C01812=1027.852,290.719,373.173,170.734,46.693,159.011
C01813=1027.858,290.967,373.141,170.739,46.692,159.011
C01814=1027.865,291.215,373.110,170.743,46.691,159.011
C01815=1027.872,291.462,373.078,170.747,46.690,159.011
C01816=1027.883,291.868,373.026,170.754,46.689,159.012
C01817=1027.894,292.273,372.973,170.761,46.687,159.012
C01818=1027.906,292.679,372.921,170.769,46.685,159.013
C01819=1027.917,293.084,372.868,170.776,46.684,159.014
C01820=1027.923,293.332,372.837,170.781,46.683,159.014
C01821=1027.930,293.579,372.804,170.785,46.682,159.014
C01822=1027.937,293.828,372.772,170.789,46.681,159.015
C01823=1027.944,294.075,372.740,170.794,46.680,159.015
C01824=1027.950,294.323,372.707,170.798,46.679,159.015
C01825=1027.957,294.571,372.676,170.803,46.679,159.016
C01826=1027.963,294.818,372.643,170.807,46.678,159.016
C01827=1027.970,295.066,372.610,170.812,46.677,159.016
C01828=1027.977,295.314,372.578,170.816,46.676,159.017
C01829=1027.983,295.562,372.546,170.821,46.675,159.017
C01830=1027.990,295.810,372.513,170.826,46.675,159.018
C01831=1027.997,296.058,372.481,170.830,46.674,159.018
C01832=1028.003,296.305,372.448,170.834,46.673,159.018
C01833=1028.010,296.553,372.415,170.838,46.672,159.019
C01834=1028.017,296.800,372.383,170.844,46.671,159.019
C01835=1028.024,297.048,372.350,170.848,46.671,159.019
C01836=1028.030,297.297,372.318,170.852,46.670,159.020
C01837=1028.037,297.544,372.286,170.857,46.669,159.020
C01838=1028.043,297.791,372.253,170.861,46.668,159.020
C01839=1028.050,298.040,372.220,170.866,46.668,159.021
C01840=1028.057,298.287,372.188,170.871,46.667,159.021
C01841=1028.063,298.535,372.155,170.875,46.666,159.022
C01842=1028.070,298.783,372.122,170.879,46.666,159.022
C01843=1028.077,299.030,372.090,170.885,46.665,159.023
C01844=1028.083,299.278,372.057,170.889,46.665,159.023
C01845=1028.090,299.526,372.024,170.893,46.663,159.023
C01846=1028.097,299.773,371.992,170.898,46.663,159.024
C01847=1028.104,300.021,371.959,170.903,46.662,159.024
C01848=1028.111,300.269,371.926,170.908,46.661,159.024
C01849=1028.118,300.517,371.894,170.912,46.661,159.025
C01850=1028.125,300.764,371.860,170.917,46.660,159.025
C01851=1028.131,301.012,371.827,170.922,46.659,159.026
C01852=1028.138,301.259,371.795,170.926,46.659,159.026
C01853=1028.145,301.507,371.762,170.930,46.658,159.026
C01854=1028.151,301.755,371.729,170.936,46.657,159.027
C01855=1028.159,302.003,371.697,170.940,46.657,159.027
C01856=1028.165,302.251,371.664,170.945,46.656,159.028
C01857=1028.172,302.498,371.630,170.950,46.656,159.028
C01858=1028.179,302.746,371.597,170.954,46.655,159.029
C01859=1028.186,302.994,371.565,170.959,46.654,159.029
C01860=1028.193,303.241,371.532,170.963,46.654,159.029
C01861=1028.200,303.489,371.498,170.969,46.653,159.030
C01862=1028.207,303.736,371.466,170.973,46.652,159.030
C01863=1028.214,303.985,371.433,170.978,46.652,159.031
C01864=1028.220,304.232,371.399,170.983,46.651,159.031
C01865=1028.228,304.480,371.367,170.987,46.651,159.032
C01866=1028.234,304.727,371.334,170.992,46.650,159.032
C01867=1028.241,304.975,371.300,170.996,46.649,159.032
C01868=1028.249,305.222,371.268,171.002,46.648,159.033
C01869=1028.255,305.470,371.235,171.006,46.648,159.033
C01870=1028.263,305.718,371.201,171.011,46.647,159.034
C01871=1028.269,305.966,371.169,171.016,46.647,159.034
C01872=1028.275,306.176,371.140,171.020,46.646,159.035
C01873=1028.281,306.388,371.112,171.024,46.646,159.035
C01874=1028.287,306.599,371.083,171.029,46.646,159.036
C01875=1028.293,306.810,371.056,171.032,46.645,159.036
C01876=1028.300,307.022,371.027,171.036,46.644,159.036
C01877=1028.305,307.233,370.999,171.040,46.644,159.037
C01878=1028.312,307.445,370.970,171.045,46.644,159.037
C01879=1028.318,307.656,370.943,171.049,46.643,159.037
C01880=1028.325,307.904,370.909,171.053,46.643,159.038
C01881=1028.331,308.151,370.876,171.059,46.642,159.038
C01882=1028.339,308.398,370.843,171.063,46.642,159.039
C01883=1028.346,308.647,370.810,171.068,46.641,159.039
C01884=1028.353,308.894,370.776,171.073,46.641,159.040
C01885=1028.360,309.141,370.742,171.078,46.640,159.040
C01886=1028.367,309.389,370.710,171.083,46.640,159.041
C01887=1028.375,309.637,370.676,171.088,46.639,159.041
C01888=1028.381,309.884,370.643,171.092,46.639,159.042
C01889=1028.388,310.132,370.610,171.098,46.638,159.042
C01890=1028.396,310.380,370.576,171.102,46.638,159.043
C01891=1028.403,310.627,370.542,171.107,46.637,159.043
C01892=1028.410,310.875,370.510,171.112,46.637,159.044
C01893=1028.417,311.123,370.476,171.117,46.636,159.044
C01894=1028.424,311.370,370.442,171.122,46.636,159.045
C01895=1028.430,311.618,370.408,171.127,46.636,159.045
C01896=1028.437,311.865,370.374,171.132,46.635,159.046
C01897=1028.444,312.113,370.340,171.137,46.635,159.046
C01898=1028.451,312.361,370.307,171.142,46.635,159.047
C01899=1028.458,312.607,370.272,171.147,46.635,159.047
C01900=1028.465,312.855,370.238,171.151,46.634,159.048
C01901=1028.472,313.103,370.204,171.157,46.634,159.049
C01902=1028.478,313.351,370.170,171.161,46.634,159.049
C01903=1028.486,313.598,370.136,171.167,46.634,159.050
C01904=1028.492,313.845,370.102,171.171,46.633,159.050
C01905=1028.499,314.093,370.068,171.177,46.633,159.051
C01906=1028.506,314.341,370.034,171.181,46.633,159.051
C01907=1028.513,314.588,369.999,171.187,46.633,159.052
C01908=1028.520,314.836,369.965,171.192,46.633,159.052
C01909=1028.526,315.083,369.932,171.197,46.632,159.053
C01910=1028.533,315.331,369.897,171.202,46.633,159.054
C01911=1028.540,315.578,369.863,171.207,46.632,159.054
C01912=1028.548,315.826,369.829,171.213,46.632,159.055
C01913=1028.554,316.074,369.795,171.217,46.632,159.055
C01914=1028.561,316.321,369.761,171.223,46.631,159.056
C01915=1028.569,316.568,369.726,171.227,46.631,159.056
C01916=1028.575,316.816,369.692,171.233,46.631,159.057
C01917=1028.582,317.064,369.658,171.237,46.631,159.057
C01918=1028.590,317.311,369.623,171.243,46.631,159.058
C01919=1028.596,317.559,369.589,171.248,46.631,159.059
C01920=1028.604,317.806,369.554,171.253,46.630,159.059
C01921=1028.611,318.053,369.521,171.258,46.630,159.060
C01922=1028.617,318.301,369.487,171.263,46.630,159.060
C01923=1028.624,318.548,369.452,171.269,46.630,159.061
C01924=1028.632,318.797,369.417,171.273,46.630,159.062
C01925=1028.639,319.044,369.383,171.279,46.630,159.062
C01926=1028.646,319.292,369.349,171.284,46.630,159.063
C01927=1028.653,319.539,369.314,171.289,46.630,159.063
C01928=1028.660,319.787,369.280,171.294,46.629,159.064
C01929=1028.668,320.034,369.245,171.300,46.629,159.065
C01930=1028.674,320.282,369.211,171.304,46.629,159.065
C01931=1028.682,320.529,369.176,171.310,46.629,159.066
C01932=1028.688,320.743,369.146,171.315,46.629,159.066
C01933=1028.694,320.957,369.116,171.319,46.629,159.067
C01934=1028.700,321.170,369.087,171.324,46.629,159.068
C01935=1028.706,321.384,369.057,171.328,46.629,159.068
C01936=1028.712,321.597,369.027,171.333,46.629,159.069
C01937=1028.719,321.811,368.997,171.337,46.629,159.069
C01938=1028.725,322.025,368.967,171.342,46.629,159.070
C01939=1028.731,322.239,368.937,171.346,46.629,159.070
C01940=1028.739,322.486,368.903,171.352,46.629,159.071
C01941=1028.746,322.733,368.868,171.356,46.629,159.071
C01942=1028.753,322.981,368.834,171.362,46.629,159.072
C01943=1028.760,323.229,368.799,171.368,46.629,159.073
C01944=1028.767,323.477,368.764,171.373,46.629,159.073
C01945=1028.775,323.724,368.729,171.378,46.629,159.074
C01946=1028.782,323.971,368.695,171.384,46.629,159.075
C01947=1028.789,324.219,368.660,171.389,46.629,159.075
C01948=1028.797,324.466,368.625,171.394,46.629,159.076
C01949=1028.804,324.714,368.590,171.399,46.629,159.077
C01950=1028.811,324.961,368.555,171.405,46.629,159.077
C01951=1028.819,325.209,368.521,171.411,46.629,159.078
C01952=1028.826,325.456,368.485,171.415,46.629,159.079
C01953=1028.834,325.703,368.451,171.421,46.629,159.079
C01954=1028.841,325.951,368.415,171.427,46.629,159.080
C01955=1028.849,326.198,368.381,171.433,46.629,159.081
C01956=1028.855,326.446,368.346,171.437,46.629,159.081
C01957=1028.863,326.693,368.311,171.443,46.629,159.082
C01958=1028.871,326.940,368.276,171.448,46.629,159.083
C01959=1028.878,327.188,368.241,171.454,46.629,159.083
C01960=1028.886,327.435,368.206,171.459,46.630,159.084
C01961=1028.893,327.683,368.171,171.465,46.630,159.085
C01962=1028.900,327.931,368.136,171.470,46.630,159.085
C01963=1028.907,328.178,368.101,171.476,46.630,159.086
C01964=1028.915,328.425,368.065,171.481,46.630,159.087
C01965=1028.922,328.673,368.030,171.486,46.630,159.087
C01966=1028.929,328.920,367.995,171.492,46.631,159.088
C01967=1028.936,329.167,367.959,171.498,46.631,159.089
C01968=1028.943,329.415,367.923,171.503,46.632,159.090
C01969=1028.951,329.662,367.889,171.509,46.632,159.090
C01970=1028.958,329.909,367.852,171.515,46.632,159.091
C01971=1028.965,330.157,367.817,171.520,46.632,159.092
C01972=1028.973,330.404,367.781,171.526,46.632,159.093
C01973=1028.980,330.652,367.746,171.531,46.633,159.093
C01974=1028.987,330.899,367.710,171.537,46.633,159.094
C01975=1028.994,331.146,367.675,171.542,46.633,159.095
C01976=1029.002,331.394,367.639,171.548,46.634,159.096
C01977=1029.009,331.641,367.604,171.554,46.633,159.096
C01978=1029.017,331.888,367.568,171.559,46.634,159.097
C01979=1029.024,332.136,367.532,171.565,46.635,159.098
C01980=1029.031,332.383,367.496,171.570,46.635,159.099
C01981=1029.038,332.631,367.461,171.576,46.635,159.100
C01982=1029.046,332.878,367.425,171.582,46.636,159.100
C01983=1029.054,333.124,367.390,171.588,46.636,159.101
C01984=1029.061,333.372,367.354,171.593,46.636,159.102
C01985=1029.069,333.620,367.318,171.599,46.637,159.103
C01986=1029.076,333.867,367.282,171.604,46.637,159.103
C01987=1029.083,334.115,367.247,171.610,46.637,159.104
C01988=1029.091,334.362,367.210,171.616,46.638,159.105
C01989=1029.098,334.609,367.175,171.622,46.638,159.106
C01990=1029.105,334.856,367.138,171.627,46.639,159.106
C01991=1029.113,335.103,367.102,171.633,46.639,159.107
C01992=1029.119,335.315,367.071,171.638,46.640,159.108
C01993=1029.125,335.527,367.041,171.643,46.640,159.109
C01994=1029.131,335.738,367.009,171.648,46.641,159.109
C01995=1029.137,335.950,366.978,171.653,46.641,159.110
C01996=1029.144,336.162,366.948,171.658,46.642,159.111
C01997=1029.150,336.372,366.916,171.662,46.642,159.111
C01998=1029.156,336.584,366.886,171.668,46.642,159.112
C01999=1029.163,336.796,366.855,171.673,46.642,159.113
C02000=1029.170,337.043,366.818,171.679,46.643,159.114
C02001=1029.178,337.290,366.782,171.685,46.643,159.115
C02002=1029.185,337.537,366.746,171.690,46.644,159.115
C02003=1029.193,337.785,366.710,171.696,46.645,159.116
C02004=1029.200,338.032,366.674,171.701,46.645,159.117
C02005=1029.208,338.279,366.638,171.707,46.646,159.118
C02006=1029.215,338.527,366.601,171.713,46.646,159.119
C02007=1029.222,338.774,366.565,171.719,46.647,159.120
C02008=1029.230,339.022,366.528,171.725,46.648,159.121
C02009=1029.238,339.269,366.491,171.731,46.648,159.121
C02010=1029.245,339.515,366.456,171.737,46.649,159.122
C02011=1029.253,339.763,366.419,171.743,46.649,159.123
C02012=1029.260,340.010,366.383,171.749,46.650,159.124
C02013=1029.268,340.257,366.346,171.755,46.650,159.125
C02014=1029.275,340.505,366.309,171.761,46.651,159.126
C02015=1029.283,340.752,366.273,171.767,46.652,159.127
C02016=1029.291,340.999,366.236,171.773,46.653,159.128
C02017=1029.297,341.246,366.200,171.779,46.653,159.128
C02018=1029.305,341.493,366.163,171.785,46.654,159.129
C02019=1029.313,341.740,366.127,171.791,46.655,159.130
C02020=1029.320,341.987,366.089,171.797,46.655,159.131
C02021=1029.328,342.235,366.053,171.803,46.656,159.132
C02022=1029.335,342.482,366.015,171.809,46.657,159.133
C02023=1029.343,342.730,365.979,171.815,46.657,159.134
C02024=1029.351,342.976,365.942,171.822,46.658,159.135
C02025=1029.358,343.223,365.905,171.827,46.659,159.136
C02026=1029.366,343.471,365.868,171.834,46.660,159.137
C02027=1029.373,343.718,365.831,171.840,46.661,159.138
C02028=1029.381,343.965,365.794,171.846,46.662,159.139
C02029=1029.389,344.212,365.758,171.852,46.662,159.139
C02030=1029.396,344.459,365.720,171.858,46.663,159.140
C02031=1029.404,344.706,365.683,171.864,46.664,159.141
C02032=1029.411,344.953,365.646,171.870,46.665,159.142
C02033=1029.419,345.201,365.610,171.876,46.665,159.143
C02034=1029.426,345.448,365.572,171.882,46.666,159.144
C02035=1029.434,345.695,365.535,171.889,46.668,159.145
C02036=1029.441,345.942,365.498,171.895,46.668,159.146
C02037=1029.450,346.189,365.460,171.901,46.669,159.147
C02038=1029.457,346.437,365.423,171.908,46.670,159.148
C02039=1029.465,346.683,365.386,171.914,46.671,159.149
C02040=1029.472,346.931,365.348,171.920,46.672,159.150
C02041=1029.480,347.177,365.311,171.926,46.673,159.151
C02042=1029.488,347.425,365.274,171.932,46.673,159.152
C02043=1029.496,347.672,365.237,171.939,46.674,159.153
C02044=1029.503,347.919,365.199,171.945,46.675,159.154
C02045=1029.511,348.166,365.162,171.951,46.677,159.155
C02046=1029.519,348.413,365.125,171.958,46.677,159.156
C02047=1029.527,348.660,365.088,171.964,46.678,159.157
C02048=1029.534,348.908,365.050,171.970,46.679,159.158
C02049=1029.542,349.154,365.011,171.977,46.680,159.159
C02050=1029.550,349.401,364.975,171.983,46.681,159.160
C02051=1029.557,349.648,364.937,171.989,46.682,159.161
C02052=1029.563,349.858,364.905,171.995,46.683,159.162
C02053=1029.570,350.068,364.873,172.000,46.684,159.163
C02054=1029.577,350.279,364.840,172.006,46.685,159.164
C02055=1029.584,350.488,364.809,172.011,46.686,159.165
C02056=1029.590,350.699,364.776,172.016,46.687,159.165
C02057=1029.597,350.908,364.745,172.023,46.688,159.166
C02058=1029.603,351.118,364.712,172.027,46.689,159.167
C02059=1029.610,351.328,364.680,172.034,46.690,159.168
C02060=1029.618,351.576,364.642,172.040,46.691,159.169
C02061=1029.625,351.822,364.604,172.046,46.692,159.170
C02062=1029.633,352.069,364.567,172.052,46.693,159.171
C02063=1029.641,352.316,364.529,172.059,46.694,159.172
C02064=1029.649,352.563,364.491,172.066,46.695,159.173
C02065=1029.656,352.810,364.453,172.072,46.696,159.174
C02066=1029.665,353.057,364.415,172.079,46.698,159.176
C02067=1029.672,353.304,364.377,172.085,46.699,159.177
C02068=1029.680,353.551,364.339,172.092,46.700,159.178
C02069=1029.688,353.798,364.301,172.098,46.701,159.179
C02070=1029.696,354.045,364.263,172.105,46.702,159.180
C02071=1029.704,354.292,364.225,172.112,46.703,159.181
C02072=1029.712,354.539,364.186,172.118,46.704,159.182
C02073=1029.720,354.786,364.149,172.125,46.706,159.183
C02074=1029.728,355.033,364.110,172.131,46.707,159.184
C02075=1029.736,355.279,364.073,172.138,46.708,159.185
C02076=1029.744,355.527,364.034,172.145,46.710,159.187
C02077=1029.752,355.773,363.996,172.151,46.711,159.188
C02078=1029.760,356.020,363.957,172.159,46.712,159.189
C02079=1029.767,356.267,363.919,172.165,46.713,159.190
C02080=1029.776,356.514,363.880,172.171,46.715,159.191
C02081=1029.784,356.761,363.842,172.179,46.716,159.192
C02082=1029.791,357.008,363.803,172.185,46.717,159.193
C02083=1029.799,357.255,363.765,172.191,46.718,159.194
C02084=1029.807,357.501,363.727,172.199,46.720,159.196
C02085=1029.815,357.749,363.688,172.206,46.721,159.197
C02086=1029.823,357.996,363.649,172.213,46.722,159.198
C02087=1029.831,358.242,363.611,172.219,46.724,159.199
C02088=1029.839,358.490,363.573,172.226,46.726,159.200
C02089=1029.847,358.737,363.534,172.233,46.726,159.202
C02090=1029.855,358.983,363.495,172.240,46.728,159.203
C02091=1029.863,359.230,363.456,172.247,46.730,159.204
C02092=1029.871,359.477,363.418,172.254,46.731,159.205
C02093=1029.879,359.724,363.379,172.260,46.732,159.206
C02094=1029.887,359.970,363.340,172.268,46.734,159.208
C02095=1029.895,360.218,363.302,172.274,46.735,159.209
C02096=1029.904,360.464,363.262,172.282,46.737,159.210
C02097=1029.912,360.711,363.224,172.288,46.738,159.211
C02098=1029.920,360.958,363.185,172.296,46.740,159.212
C02099=1029.927,361.205,363.145,172.302,46.741,159.214
C02100=1029.935,361.452,363.107,172.310,46.743,159.215
C02101=1029.944,361.699,363.068,172.316,46.745,159.216
C02102=1029.952,361.945,363.028,172.323,46.746,159.217
C02103=1029.959,362.192,362.989,172.330,46.748,159.219
C02104=1029.968,362.439,362.950,172.337,46.749,159.220
C02105=1029.976,362.685,362.911,172.344,46.751,159.221
C02106=1029.983,362.933,362.871,172.351,46.752,159.222
C02107=1029.992,363.179,362.832,172.359,46.754,159.224
C02108=1030.000,363.426,362.793,172.365,46.756,159.225
C02109=1030.008,363.673,362.753,172.373,46.757,159.226
C02110=1030.016,363.920,362.714,172.380,46.759,159.228
C02111=1030.025,364.167,362.675,172.387,46.760,159.229
C02112=1030.032,364.379,362.641,172.394,46.762,159.230
C02113=1030.038,364.592,362.607,172.400,46.763,159.231
C02114=1030.046,364.805,362.572,172.405,46.765,159.232
C02115=1030.053,365.019,362.539,172.412,46.766,159.233
C02116=1030.060,365.232,362.505,172.418,46.768,159.234
C02117=1030.067,365.445,362.471,172.425,46.769,159.236
C02118=1030.075,365.658,362.436,172.431,46.770,159.237
C02119=1030.081,365.871,362.402,172.437,46.772,159.238
C02120=1030.089,366.118,362.363,172.444,46.774,159.239
C02121=1030.098,366.364,362.323,172.452,46.776,159.241
C02122=1030.106,366.611,362.283,172.458,46.777,159.242
C02123=1030.114,366.858,362.244,172.466,46.779,159.243
C02124=1030.123,367.104,362.205,172.474,46.781,159.245
C02125=1030.131,367.352,362.165,172.481,46.783,159.246
C02126=1030.140,367.598,362.124,172.488,46.784,159.247
C02127=1030.148,367.845,362.085,172.496,46.786,159.249
C02128=1030.156,368.092,362.045,172.503,46.788,159.250
C02129=1030.164,368.338,362.006,172.510,46.790,159.251
C02130=1030.173,368.584,361.966,172.518,46.792,159.253
C02131=1030.181,368.832,361.926,172.525,46.794,159.254
C02132=1030.190,369.078,361.886,172.533,46.796,159.256
C02133=1030.199,369.324,361.846,172.541,46.798,159.257
C02134=1030.206,369.571,361.806,172.548,46.800,159.258
C02135=1030.214,369.817,361.766,172.555,46.801,159.260
C02136=1030.223,370.065,361.726,172.563,46.803,159.261
C02137=1030.231,370.311,361.685,172.571,46.805,159.263
C02138=1030.239,370.558,361.645,172.578,46.807,159.264
C02139=1030.248,370.804,361.605,172.585,46.809,159.265
C02140=1030.256,371.051,361.564,172.593,46.811,159.267
C02141=1030.265,371.297,361.525,172.601,46.813,159.268
C02142=1030.273,371.544,361.484,172.608,46.815,159.270
C02143=1030.282,371.791,361.443,172.616,46.817,159.271
C02144=1030.290,372.037,361.403,172.624,46.819,159.273
C02145=1030.298,372.283,361.363,172.632,46.821,159.274
C02146=1030.307,372.531,361.322,172.639,46.823,159.276
C02147=1030.315,372.777,361.282,172.646,46.825,159.277
C02148=1030.323,373.023,361.242,172.654,46.827,159.279
C02149=1030.332,373.270,361.201,172.662,46.829,159.280
C02150=1030.341,373.516,361.161,172.670,46.832,159.282
C02151=1030.350,373.763,361.120,172.678,46.834,159.283
C02152=1030.358,374.009,361.079,172.686,46.836,159.285
C02153=1030.367,374.256,361.039,172.694,46.838,159.286
C02154=1030.375,374.502,360.998,172.701,46.841,159.288
C02155=1030.384,374.749,360.957,172.709,46.843,159.289
C02156=1030.392,374.995,360.917,172.717,46.844,159.291
C02157=1030.401,375.242,360.876,172.724,46.846,159.292
C02158=1030.409,375.488,360.835,172.733,46.849,159.294
C02159=1030.418,375.735,360.795,172.741,46.851,159.295
C02160=1030.427,375.981,360.754,172.749,46.853,159.297
C02161=1030.435,376.228,360.713,172.757,46.855,159.298
C02162=1030.445,376.474,360.672,172.765,46.858,159.300
C02163=1030.453,376.721,360.632,172.773,46.860,159.301
C02164=1030.462,376.967,360.590,172.781,46.862,159.303
C02165=1030.471,377.214,360.549,172.789,46.864,159.305
C02166=1030.479,377.460,360.509,172.797,46.867,159.306
C02167=1030.488,377.706,360.467,172.805,46.869,159.308
C02168=1030.497,377.953,360.426,172.813,46.871,159.309
C02169=1030.505,378.199,360.385,172.821,46.874,159.311
C02170=1030.514,378.445,360.343,172.829,46.876,159.313
C02171=1030.522,378.692,360.302,172.837,46.878,159.314
C02172=1030.530,378.915,360.265,172.844,46.881,159.316
C02173=1030.538,379.139,360.227,172.852,46.883,159.317
C02174=1030.546,379.363,360.189,172.859,46.885,159.319
C02175=1030.553,379.586,360.152,172.867,46.887,159.320
C02176=1030.561,379.810,360.114,172.874,46.890,159.322
C02177=1030.570,380.034,360.076,172.882,46.892,159.323
C02178=1030.578,380.258,360.039,172.889,46.894,159.325
C02179=1030.586,380.480,360.001,172.897,46.896,159.326
C02180=1030.594,380.727,359.960,172.905,46.899,159.328
C02181=1030.603,380.974,359.918,172.913,46.901,159.330
C02182=1030.612,381.220,359.876,172.921,46.904,159.331
C02183=1030.621,381.466,359.835,172.930,46.906,159.333
C02184=1030.630,381.713,359.793,172.938,46.909,159.334
C02185=1030.639,381.959,359.751,172.947,46.911,159.336
C02186=1030.647,382.206,359.709,172.955,46.914,159.338
C02187=1030.656,382.452,359.667,172.963,46.916,159.340
C02188=1030.665,382.699,359.625,172.972,46.919,159.341
C02189=1030.674,382.944,359.583,172.980,46.922,159.343
C02190=1030.683,383.191,359.541,172.989,46.924,159.345
C02191=1030.692,383.437,359.500,172.997,46.926,159.346
C02192=1030.701,383.683,359.458,173.006,46.929,159.348
C02193=1030.710,383.930,359.416,173.014,46.932,159.350
C02194=1030.719,384.175,359.374,173.023,46.934,159.352
C02195=1030.728,384.422,359.332,173.032,46.937,159.354
C02196=1030.737,384.668,359.290,173.040,46.940,159.355
C02197=1030.746,384.914,359.248,173.048,46.943,159.357
C02198=1030.755,385.160,359.206,173.058,46.945,159.359
C02199=1030.765,385.406,359.164,173.066,46.948,159.361
C02200=1030.774,385.652,359.122,173.074,46.950,159.362
C02201=1030.783,385.899,359.079,173.084,46.953,159.364
C02202=1030.792,386.145,359.038,173.092,46.956,159.366
C02203=1030.802,386.391,358.995,173.101,46.959,159.368
C02204=1030.810,386.637,358.953,173.110,46.962,159.370
C02205=1030.820,386.884,358.911,173.118,46.964,159.371
C02206=1030.829,387.130,358.868,173.128,46.967,159.373
C02207=1030.838,387.376,358.826,173.136,46.970,159.375
C02208=1030.847,387.622,358.783,173.145,46.973,159.377
C02209=1030.857,387.868,358.741,173.154,46.976,159.379
C02210=1030.865,388.114,358.698,173.163,46.979,159.381
C02211=1030.875,388.360,358.655,173.172,46.981,159.383
C02212=1030.884,388.607,358.612,173.181,46.985,159.384
C02213=1030.893,388.853,358.569,173.189,46.988,159.386
C02214=1030.902,389.098,358.527,173.199,46.990,159.388
C02215=1030.912,389.345,358.484,173.207,46.993,159.390
C02216=1030.920,389.591,358.441,173.217,46.996,159.392
C02217=1030.930,389.837,358.399,173.225,46.999,159.394
C02218=1030.940,390.083,358.356,173.235,47.002,159.396
C02219=1030.948,390.329,358.313,173.243,47.005,159.398
C02220=1030.958,390.576,358.270,173.253,47.008,159.400
C02221=1030.967,390.821,358.226,173.262,47.011,159.402
C02222=1030.977,391.067,358.183,173.271,47.014,159.404
C02223=1030.985,391.314,358.140,173.281,47.017,159.406
C02224=1030.995,391.559,358.097,173.289,47.020,159.408
C02225=1031.004,391.805,358.054,173.299,47.023,159.409
C02226=1031.014,392.052,358.011,173.308,47.027,159.412
C02227=1031.023,392.297,357.968,173.317,47.029,159.413
C02228=1031.032,392.544,357.925,173.327,47.033,159.416
C02229=1031.042,392.790,357.881,173.336,47.036,159.417
C02230=1031.051,393.036,357.838,173.345,47.039,159.420
C02231=1031.061,393.281,357.794,173.355,47.042,159.421
C02232=1031.071,393.545,357.748,173.365,47.046,159.424
C02233=1031.081,393.811,357.701,173.375,47.049,159.426
C02234=1031.092,394.074,357.655,173.385,47.052,159.428
C02235=1031.101,394.338,357.608,173.395,47.056,159.430
C02236=1031.111,394.584,357.563,173.405,47.060,159.432
C02237=1031.121,394.830,357.520,173.414,47.062,159.434
C02238=1031.130,395.076,357.476,173.424,47.066,159.436
C02239=1031.139,395.322,357.433,173.433,47.069,159.439
C02240=1031.149,395.568,357.389,173.443,47.072,159.441
C02241=1031.158,395.814,357.345,173.453,47.076,159.443
C02242=1031.168,396.061,357.301,173.462,47.079,159.445
C02243=1031.178,396.306,357.257,173.471,47.083,159.447
C02244=1031.187,396.551,357.213,173.481,47.086,159.449
C02245=1031.197,396.797,357.169,173.491,47.089,159.451
C02246=1031.207,397.043,357.125,173.501,47.093,159.454
C02247=1031.216,397.289,357.081,173.511,47.096,159.456
C02248=1031.225,397.521,357.040,173.520,47.099,159.457
C02249=1031.235,397.753,356.998,173.529,47.103,159.460
C02250=1031.244,397.986,356.956,173.538,47.106,159.462
C02251=1031.253,398.218,356.915,173.548,47.109,159.464
C02252=1031.262,398.450,356.873,173.557,47.112,159.466
C02253=1031.271,398.682,356.831,173.566,47.116,159.468
C02254=1031.280,398.914,356.790,173.576,47.119,159.470
C02255=1031.290,399.145,356.747,173.585,47.122,159.472
C02256=1031.300,399.392,356.703,173.595,47.126,159.474
C02257=1031.309,399.637,356.658,173.605,47.130,159.476
C02258=1031.319,399.883,356.614,173.615,47.133,159.479
C02259=1031.329,400.128,356.570,173.625,47.137,159.481
C02260=1031.339,400.374,356.525,173.635,47.140,159.483
C02261=1031.348,400.620,356.481,173.646,47.144,159.486
C02262=1031.359,400.866,356.436,173.655,47.147,159.488
C02263=1031.368,401.112,356.391,173.666,47.151,159.490
C02264=1031.378,401.357,356.346,173.676,47.155,159.492
C02265=1031.388,401.603,356.302,173.686,47.159,159.495
C02266=1031.398,401.849,356.256,173.697,47.162,159.497
C02267=1031.408,402.095,356.211,173.707,47.166,159.499
C02268=1031.417,402.340,356.167,173.717,47.170,159.502
C02269=1031.427,402.586,356.122,173.728,47.174,159.504
C02270=1031.438,402.832,356.077,173.738,47.178,159.506
C02271=1031.447,403.077,356.032,173.748,47.182,159.509
C02272=1031.457,403.323,355.987,173.759,47.185,159.511
C02273=1031.468,403.568,355.941,173.769,47.189,159.513
C02274=1031.477,403.814,355.896,173.779,47.193,159.516
C02275=1031.488,404.060,355.851,173.790,47.197,159.518
C02276=1031.498,404.305,355.806,173.800,47.201,159.521
C02277=1031.507,404.551,355.761,173.811,47.204,159.523
C02278=1031.518,404.797,355.716,173.822,47.209,159.525
C02279=1031.527,405.042,355.669,173.832,47.212,159.528
C02280=1031.537,405.288,355.624,173.843,47.216,159.530
C02281=1031.548,405.534,355.578,173.854,47.220,159.533
C02282=1031.558,405.779,355.533,173.864,47.224,159.535
C02283=1031.568,406.025,355.488,173.875,47.228,159.538
C02284=1031.578,406.270,355.442,173.886,47.232,159.540
C02285=1031.589,406.516,355.397,173.896,47.236,159.542
C02286=1031.599,406.762,355.351,173.908,47.240,159.545
C02287=1031.609,407.006,355.305,173.918,47.245,159.548
C02288=1031.619,407.252,355.259,173.929,47.248,159.550
C02289=1031.629,407.499,355.214,173.940,47.252,159.553
C02290=1031.640,407.744,355.168,173.951,47.256,159.555
C02291=1031.650,407.989,355.122,173.962,47.261,159.558
C02292=1031.661,408.247,355.074,173.973,47.265,159.560
C02293=1031.672,408.505,355.026,173.985,47.269,159.563
C02294=1031.683,408.763,354.977,173.997,47.273,159.566
C02295=1031.694,409.021,354.929,174.009,47.278,159.568
C02296=1031.705,409.267,354.883,174.019,47.282,159.571
C02297=1031.716,409.512,354.837,174.031,47.286,159.574
C02298=1031.727,409.757,354.791,174.042,47.290,159.576
C02299=1031.736,410.003,354.744,174.053,47.295,159.579
C02300=1031.747,410.249,354.698,174.065,47.299,159.581
C02301=1031.758,410.495,354.652,174.076,47.303,159.584
C02302=1031.769,410.740,354.606,174.087,47.308,159.587
C02303=1031.778,410.985,354.559,174.098,47.312,159.589
C02304=1031.789,411.230,354.513,174.110,47.317,159.592
C02305=1031.799,411.476,354.466,174.121,47.321,159.595
C02306=1031.810,411.721,354.420,174.133,47.326,159.598
C02307=1031.821,411.966,354.373,174.144,47.329,159.600
C02308=1031.831,412.212,354.327,174.156,47.334,159.603
C02309=1031.842,412.457,354.280,174.167,47.339,159.606
C02310=1031.853,412.703,354.232,174.179,47.343,159.608
C02311=1031.864,412.948,354.186,174.190,47.347,159.611
C02312=1031.874,413.194,354.139,174.202,47.352,159.614
C02313=1031.884,413.439,354.093,174.214,47.356,159.617
C02314=1031.895,413.685,354.045,174.226,47.361,159.619
C02315=1031.906,413.930,353.998,174.238,47.366,159.622
C02316=1031.916,414.175,353.951,174.249,47.370,159.625
C02317=1031.927,414.420,353.905,174.261,47.375,159.628
C02318=1031.939,414.666,353.858,174.272,47.379,159.631
C02319=1031.949,414.911,353.810,174.284,47.384,159.633
C02320=1031.961,415.156,353.763,174.296,47.388,159.636
C02321=1031.971,415.401,353.715,174.308,47.393,159.639
C02322=1031.983,415.647,353.668,174.320,47.398,159.642
C02323=1031.993,415.892,353.621,174.333,47.402,159.645
C02324=1032.005,416.138,353.573,174.345,47.407,159.648
C02325=1032.015,416.383,353.526,174.357,47.412,159.651
C02326=1032.026,416.628,353.479,174.369,47.417,159.654
C02327=1032.037,416.874,353.431,174.381,47.421,159.657
C02328=1032.048,417.118,353.383,174.394,47.426,159.660
C02329=1032.059,417.364,353.336,174.405,47.431,159.662
C02330=1032.070,417.609,353.288,174.419,47.436,159.665
C02331=1032.081,417.854,353.240,174.431,47.441,159.668
C02332=1032.092,418.100,353.192,174.443,47.446,159.671
C02333=1032.103,418.345,353.145,174.455,47.451,159.675
C02334=1032.114,418.590,353.097,174.468,47.456,159.678
C02335=1032.125,418.835,353.048,174.481,47.460,159.681
C02336=1032.137,419.080,353.001,174.493,47.465,159.684
C02337=1032.148,419.325,352.953,174.505,47.470,159.687
C02338=1032.159,419.570,352.904,174.518,47.475,159.690
C02339=1032.170,419.816,352.856,174.531,47.480,159.693
C02340=1032.182,420.061,352.808,174.544,47.485,159.696
C02341=1032.193,420.306,352.760,174.556,47.490,159.699
C02342=1032.204,420.550,352.711,174.569,47.495,159.702
C02343=1032.215,420.796,352.663,174.582,47.500,159.705
C02344=1032.227,421.041,352.615,174.594,47.506,159.708
C02345=1032.238,421.285,352.566,174.608,47.510,159.711
C02346=1032.249,421.531,352.518,174.621,47.516,159.715
C02347=1032.260,421.776,352.470,174.634,47.521,159.718
C02348=1032.272,422.020,352.421,174.647,47.526,159.721
C02349=1032.284,422.267,352.373,174.659,47.531,159.724
C02350=1032.295,422.511,352.324,174.673,47.536,159.727
C02351=1032.307,422.756,352.275,174.686,47.541,159.731
C02352=1032.319,423.025,352.222,174.700,47.547,159.734
C02353=1032.332,423.293,352.169,174.715,47.552,159.738
C02354=1032.345,423.561,352.115,174.729,47.559,159.741
C02355=1032.357,423.829,352.062,174.744,47.564,159.745
C02356=1032.369,424.073,352.013,174.757,47.570,159.748
C02357=1032.380,424.318,351.964,174.771,47.575,159.751
C02358=1032.392,424.563,351.915,174.784,47.580,159.755
C02359=1032.404,424.808,351.864,174.798,47.586,159.758
C02360=1032.415,425.052,351.815,174.812,47.591,159.762
C02361=1032.427,425.297,351.766,174.825,47.596,159.765
C02362=1032.439,425.543,351.717,174.839,47.602,159.768
C02363=1032.450,425.787,351.668,174.852,47.607,159.772
C02364=1032.463,426.032,351.618,174.866,47.613,159.775
C02365=1032.474,426.277,351.569,174.879,47.618,159.778
C02366=1032.486,426.522,351.519,174.893,47.624,159.782
C02367=1032.498,426.767,351.470,174.908,47.629,159.785
C02368=1032.510,427.011,351.420,174.922,47.635,159.789
C02369=1032.521,427.256,351.371,174.936,47.640,159.792
C02370=1032.534,427.501,351.321,174.950,47.646,159.796
C02371=1032.546,427.746,351.270,174.964,47.652,159.799
C02372=1032.557,427.990,351.220,174.977,47.657,159.803
C02373=1032.569,428.236,351.171,174.992,47.664,159.806
C02374=1032.581,428.480,351.121,175.006,47.669,159.810
C02375=1032.593,428.725,351.071,175.021,47.675,159.814
C02376=1032.605,428.969,351.021,175.035,47.680,159.817
C02377=1032.617,429.215,350.970,175.049,47.686,159.821
C02378=1032.629,429.458,350.920,175.063,47.692,159.824
C02379=1032.641,429.703,350.870,175.078,47.697,159.828
C02380=1032.654,429.948,350.820,175.092,47.704,159.832
C02381=1032.665,430.193,350.769,175.107,47.709,159.835
C02382=1032.678,430.437,350.718,175.121,47.715,159.839
C02383=1032.690,430.682,350.668,175.136,47.721,159.843
C02384=1032.702,430.927,350.618,175.151,47.727,159.846
C02385=1032.715,431.171,350.567,175.165,47.733,159.850
C02386=1032.727,431.416,350.516,175.180,47.739,159.854
C02387=1032.739,431.660,350.466,175.194,47.745,159.857
C02388=1032.752,431.904,350.415,175.210,47.751,159.861
C02389=1032.764,432.149,350.365,175.225,47.756,159.865
C02390=1032.777,432.393,350.314,175.239,47.763,159.869
C02391=1032.789,432.638,350.262,175.255,47.769,159.873
C02392=1032.801,432.882,350.212,175.270,47.775,159.877
C02393=1032.814,433.127,350.162,175.285,47.781,159.880
C02394=1032.827,433.372,350.110,175.300,47.787,159.884
C02395=1032.839,433.616,350.060,175.316,47.793,159.888
C02396=1032.851,433.861,350.008,175.331,47.799,159.892
C02397=1032.865,434.105,349.956,175.347,47.805,159.896
C02398=1032.877,434.349,349.905,175.362,47.811,159.900
C02399=1032.889,434.594,349.854,175.378,47.817,159.904
C02400=1032.903,434.838,349.803,175.392,47.824,159.908
C02401=1032.915,435.082,349.751,175.408,47.830,159.912
C02402=1032.928,435.327,349.700,175.424,47.836,159.916
C02403=1032.941,435.571,349.648,175.439,47.843,159.920
C02404=1032.953,435.816,349.596,175.455,47.849,159.924
C02405=1032.966,436.060,349.545,175.472,47.855,159.928
C02406=1032.979,436.304,349.492,175.488,47.862,159.932
C02407=1032.992,436.548,349.441,175.503,47.868,159.936
C02408=1033.004,436.793,349.389,175.519,47.874,159.940
C02409=1033.018,437.037,349.337,175.535,47.881,159.944
C02410=1033.030,437.281,349.285,175.551,47.887,159.948
C02411=1033.044,437.525,349.233,175.568,47.894,159.952
C02412=1033.057,437.782,349.178,175.585,47.900,159.957
C02413=1033.071,438.040,349.123,175.601,47.908,159.961
C02414=1033.085,438.296,349.068,175.619,47.915,159.966
C02415=1033.098,438.553,349.013,175.636,47.921,159.970
C02416=1033.111,438.798,348.961,175.653,47.928,159.974
C02417=1033.125,439.042,348.909,175.669,47.934,159.978
C02418=1033.138,439.286,348.856,175.686,47.941,159.983
C02419=1033.151,439.531,348.804,175.702,47.948,159.987
C02420=1033.164,439.775,348.751,175.719,47.954,159.991
C02421=1033.177,440.018,348.697,175.735,47.961,159.996
C02422=1033.191,440.263,348.645,175.753,47.968,160.000
C02423=1033.204,440.507,348.592,175.770,47.975,160.004
C02424=1033.217,440.751,348.539,175.786,47.982,160.009
C02425=1033.231,440.994,348.486,175.803,47.988,160.013
C02426=1033.244,441.238,348.433,175.821,47.995,160.018
C02427=1033.258,441.483,348.380,175.838,48.002,160.022
C02428=1033.272,441.727,348.327,175.855,48.009,160.027
C02429=1033.285,441.971,348.274,175.871,48.015,160.031
C02430=1033.299,442.214,348.221,175.889,48.022,160.036
C02431=1033.312,442.459,348.168,175.906,48.029,160.040
C02432=1033.325,442.703,348.114,175.924,48.037,160.045
C02433=1033.339,442.946,348.061,175.941,48.044,160.049
C02434=1033.353,443.191,348.008,175.959,48.050,160.054
C02435=1033.367,443.434,347.954,175.977,48.057,160.058
C02436=1033.381,443.677,347.900,175.995,48.064,160.063
C02437=1033.395,443.919,347.848,176.012,48.071,160.068
C02438=1033.410,444.163,347.796,176.030,48.078,160.072
C02439=1033.425,444.407,347.743,176.049,48.085,160.077
C02440=1033.441,444.650,347.692,176.066,48.092,160.081
C02441=1033.457,444.894,347.641,176.085,48.098,160.086
C02442=1033.474,445.137,347.589,176.103,48.105,160.091
C02443=1033.492,445.381,347.539,176.120,48.111,160.095
C02444=1033.509,445.625,347.489,176.138,48.117,160.099
C02445=1033.527,445.869,347.439,176.157,48.124,160.104
C02446=1033.546,446.113,347.391,176.176,48.130,160.109
C02447=1033.566,446.358,347.341,176.195,48.136,160.113
C02448=1033.586,446.602,347.293,176.213,48.142,160.117
C02449=1033.606,446.845,347.246,176.232,48.148,160.122
C02450=1033.627,447.089,347.198,176.251,48.153,160.126
C02451=1033.648,447.335,347.151,176.270,48.160,160.131
C02452=1033.671,447.579,347.105,176.289,48.165,160.135
C02453=1033.693,447.823,347.058,176.308,48.171,160.140
C02454=1033.716,448.068,347.012,176.327,48.177,160.144
C02455=1033.739,448.313,346.967,176.346,48.182,160.149
C02456=1033.764,448.558,346.922,176.365,48.187,160.153
C02457=1033.788,448.802,346.877,176.385,48.192,160.158
C02458=1033.813,449.048,346.833,176.404,48.198,160.162
C02459=1033.838,449.293,346.790,176.424,48.203,160.166
C02460=1033.865,449.537,346.747,176.444,48.208,160.171
C02461=1033.891,449.783,346.705,176.463,48.213,160.175
C02462=1033.918,450.029,346.662,176.483,48.218,160.180
C02463=1033.946,450.273,346.620,176.503,48.223,160.184
C02464=1033.974,450.519,346.578,176.523,48.228,160.188
C02465=1034.003,450.765,346.537,176.544,48.232,160.193
C02466=1034.032,451.010,346.497,176.564,48.237,160.197
C02467=1034.062,451.255,346.457,176.583,48.242,160.201
C02468=1034.092,451.500,346.417,176.604,48.246,160.206
C02469=1034.122,451.747,346.377,176.625,48.250,160.210
C02470=1034.154,451.992,346.338,176.645,48.255,160.214
C02471=1034.185,452.237,346.300,176.666,48.259,160.219
C02472=1034.231,452.584,346.246,176.695,48.266,160.225
C02473=1034.278,452.931,346.194,176.725,48.271,160.231
C02474=1033.992,452.993,345.866,176.728,48.338,160.252
C02475=1033.949,452.671,345.914,176.701,48.333,160.247
C02476=1033.905,452.348,345.964,176.673,48.328,160.241
C02477=1033.874,452.102,346.002,176.652,48.323,160.237
C02478=1033.843,451.857,346.040,176.632,48.319,160.232
C02479=1033.811,451.612,346.080,176.611,48.315,160.228
C02480=1033.781,451.365,346.119,176.591,48.310,160.224
C02481=1033.751,451.120,346.159,176.570,48.306,160.219
C02482=1033.722,450.875,346.200,176.550,48.301,160.215
C02483=1033.693,450.629,346.240,176.530,48.297,160.211
C02484=1033.664,450.384,346.281,176.510,48.292,160.206
C02485=1033.637,450.139,346.323,176.490,48.287,160.202
C02486=1033.609,449.894,346.366,176.470,48.283,160.198
C02487=1033.582,449.648,346.408,176.450,48.278,160.193
C02488=1033.556,449.403,346.450,176.430,48.273,160.189
C02489=1033.529,449.158,346.494,176.410,48.268,160.184
C02490=1033.505,448.913,346.538,176.391,48.262,160.180
C02491=1033.479,448.668,346.582,176.371,48.257,160.175
C02492=1033.455,448.423,346.627,176.352,48.252,160.171
C02493=1033.432,448.178,346.672,176.333,48.247,160.167
C02494=1033.409,447.933,346.717,176.313,48.241,160.162
C02495=1033.386,447.690,346.764,176.294,48.236,160.158
C02496=1033.363,447.444,346.810,176.275,48.231,160.153
C02497=1033.342,447.200,346.857,176.256,48.224,160.149
C02498=1033.321,446.956,346.904,176.237,48.219,160.144
C02499=1033.300,446.711,346.952,176.218,48.213,160.140
C02500=1033.279,446.468,346.999,176.200,48.207,160.135
C02501=1033.260,446.223,347.048,176.180,48.202,160.131
C02502=1033.241,445.979,347.097,176.162,48.195,160.126
C02503=1033.222,445.735,347.146,176.144,48.189,160.122
C02504=1033.204,445.492,347.196,176.125,48.183,160.117
C02505=1033.186,445.247,347.246,176.107,48.177,160.113
C02506=1033.169,445.003,347.297,176.089,48.170,160.108
C02507=1033.152,444.759,347.348,176.070,48.164,160.104
C02508=1033.136,444.517,347.399,176.053,48.157,160.099
C02509=1033.120,444.273,347.450,176.034,48.151,160.095
C02510=1033.105,444.029,347.504,176.016,48.144,160.090
C02511=1033.091,443.786,347.556,175.998,48.137,160.085
C02512=1033.077,443.544,347.609,175.981,48.130,160.081
C02513=1033.063,443.299,347.663,175.963,48.123,160.076
C02514=1033.049,443.056,347.715,175.946,48.116,160.072
C02515=1033.035,442.812,347.770,175.928,48.109,160.067
C02516=1033.022,442.568,347.823,175.910,48.103,160.063
C02517=1033.008,442.324,347.876,175.892,48.096,160.058
C02518=1032.995,442.081,347.929,175.875,48.089,160.053
C02519=1032.980,441.836,347.982,175.857,48.082,160.049
C02520=1032.967,441.592,348.036,175.841,48.076,160.045
C02521=1032.954,441.349,348.089,175.824,48.069,160.040
C02522=1032.940,441.105,348.141,175.806,48.062,160.036
C02523=1032.927,440.861,348.195,175.789,48.056,160.031
C02524=1032.913,440.616,348.248,175.772,48.049,160.027
C02525=1032.900,440.372,348.300,175.756,48.042,160.023
C02526=1032.887,440.128,348.353,175.738,48.035,160.018
C02527=1032.873,439.884,348.406,175.721,48.029,160.014
C02528=1032.860,439.640,348.458,175.705,48.022,160.009
C02529=1032.847,439.396,348.512,175.688,48.016,160.005
C02530=1032.834,439.152,348.563,175.671,48.009,160.001
C02531=1032.821,438.908,348.616,175.655,48.002,159.997
C02532=1032.808,438.664,348.668,175.638,47.996,159.992
C02533=1032.793,438.405,348.724,175.620,47.989,159.988
C02534=1032.779,438.148,348.779,175.603,47.983,159.984
C02535=1032.766,437.890,348.835,175.586,47.976,159.979
C02536=1032.753,437.631,348.889,175.569,47.969,159.975
C02537=1032.739,437.387,348.941,175.553,47.962,159.970
C02538=1032.726,437.142,348.994,175.537,47.956,159.966
C02539=1032.713,436.899,349.045,175.520,47.950,159.962
C02540=1032.701,436.654,349.098,175.504,47.943,159.958
C02541=1032.687,436.410,349.150,175.489,47.937,159.954
C02542=1032.675,436.166,349.202,175.473,47.930,159.950
C02543=1032.662,435.921,349.253,175.457,47.924,159.946
C02544=1032.650,435.677,349.305,175.440,47.918,159.942
C02545=1032.636,435.433,349.357,175.425,47.912,159.938
C02546=1032.623,435.189,349.408,175.409,47.906,159.934
C02547=1032.611,434.943,349.459,175.394,47.900,159.930
C02548=1032.598,434.700,349.511,175.378,47.893,159.926
C02549=1032.586,434.455,349.562,175.362,47.887,159.922
C02550=1032.573,434.211,349.614,175.347,47.881,159.918
C02551=1032.560,433.967,349.665,175.331,47.875,159.914
C02552=1032.547,433.722,349.717,175.317,47.869,159.910
C02553=1032.535,433.478,349.768,175.301,47.863,159.906
C02554=1032.522,433.233,349.818,175.286,47.857,159.902
C02555=1032.510,432.989,349.869,175.270,47.851,159.899
C02556=1032.496,432.744,349.920,175.255,47.845,159.895
C02557=1032.485,432.499,349.971,175.240,47.840,159.891
C02558=1032.472,432.255,350.022,175.225,47.833,159.887
C02559=1032.460,432.011,350.073,175.210,47.827,159.883
C02560=1032.447,431.766,350.123,175.195,47.822,159.880
C02561=1032.435,431.522,350.174,175.180,47.816,159.876
C02562=1032.422,431.277,350.224,175.165,47.810,159.872
C02563=1032.410,431.032,350.275,175.151,47.804,159.868
C02564=1032.398,430.788,350.326,175.135,47.798,159.865
C02565=1032.386,430.543,350.376,175.121,47.792,159.861
C02566=1032.373,430.298,350.426,175.106,47.786,159.857
C02567=1032.361,430.054,350.477,175.092,47.781,159.854
C02568=1032.349,429.809,350.528,175.077,47.775,159.850
C02569=1032.337,429.564,350.578,175.063,47.769,159.846
C02570=1032.325,429.320,350.628,175.048,47.764,159.843
C02571=1032.313,429.075,350.678,175.033,47.758,159.839
C02572=1032.300,428.831,350.728,175.020,47.752,159.836
C02573=1032.288,428.586,350.779,175.005,47.747,159.832
C02574=1032.277,428.342,350.829,174.991,47.741,159.828
C02575=1032.265,428.096,350.878,174.977,47.735,159.825
C02576=1032.252,427.852,350.928,174.963,47.730,159.821
C02577=1032.241,427.608,350.978,174.949,47.724,159.818
C02578=1032.229,427.362,351.029,174.934,47.719,159.814
C02579=1032.217,427.118,351.078,174.920,47.713,159.811
C02580=1032.205,426.873,351.128,174.906,47.707,159.807
C02581=1032.193,426.628,351.178,174.892,47.702,159.804
C02582=1032.182,426.383,351.227,174.878,47.697,159.800
C02583=1032.169,426.138,351.277,174.865,47.691,159.797
C02584=1032.158,425.894,351.326,174.851,47.686,159.794
C02585=1032.147,425.649,351.375,174.837,47.681,159.790
C02586=1032.134,425.404,351.425,174.823,47.675,159.787
C02587=1032.123,425.159,351.474,174.809,47.670,159.783
C02588=1032.111,424.914,351.524,174.796,47.665,159.780
C02589=1032.099,424.669,351.573,174.782,47.659,159.777
C02590=1032.088,424.424,351.622,174.769,47.654,159.774
C02591=1032.076,424.179,351.671,174.755,47.648,159.770
C02592=1032.064,423.935,351.719,174.742,47.643,159.767
C02593=1032.052,423.664,351.774,174.727,47.638,159.763
C02594=1032.039,423.394,351.828,174.712,47.632,159.760
C02595=1032.027,423.124,351.882,174.698,47.626,159.756
C02596=1032.014,422.854,351.936,174.683,47.620,159.752
C02597=1032.002,422.607,351.985,174.669,47.615,159.749
C02598=1031.990,422.363,352.033,174.657,47.610,159.746
C02599=1031.978,422.118,352.082,174.644,47.605,159.743
C02600=1031.967,421.873,352.130,174.630,47.600,159.740
C02601=1031.956,421.628,352.179,174.618,47.595,159.736
C02602=1031.944,421.383,352.227,174.604,47.590,159.733
C02603=1031.933,421.138,352.275,174.591,47.585,159.730
C02604=1031.922,420.893,352.324,174.579,47.580,159.727
C02605=1031.910,420.648,352.373,174.565,47.575,159.724
C02606=1031.899,420.403,352.420,174.553,47.570,159.721
C02607=1031.888,420.157,352.469,174.540,47.565,159.718
C02608=1031.876,419.912,352.518,174.527,47.560,159.715
C02609=1031.865,419.668,352.565,174.514,47.555,159.711
C02610=1031.854,419.423,352.613,174.502,47.550,159.708
C02611=1031.843,419.177,352.662,174.489,47.545,159.705
C02612=1031.832,418.932,352.710,174.476,47.541,159.702
C02613=1031.820,418.687,352.758,174.464,47.536,159.699
C02614=1031.809,418.442,352.806,174.452,47.531,159.696
C02615=1031.798,418.196,352.853,174.439,47.526,159.693
C02616=1031.787,417.951,352.901,174.427,47.521,159.690
C02617=1031.776,417.707,352.949,174.414,47.516,159.687
C02618=1031.765,417.461,352.997,174.401,47.512,159.684
C02619=1031.754,417.215,353.045,174.389,47.507,159.681
C02620=1031.743,416.971,353.092,174.377,47.502,159.678
C02621=1031.732,416.726,353.140,174.365,47.498,159.676
C02622=1031.722,416.480,353.187,174.353,47.493,159.672
C02623=1031.710,416.235,353.234,174.340,47.488,159.670
C02624=1031.699,415.989,353.283,174.328,47.483,159.667
C02625=1031.688,415.744,353.329,174.316,47.479,159.664
C02626=1031.677,415.499,353.376,174.304,47.474,159.661
C02627=1031.666,415.254,353.424,174.292,47.470,159.658
C02628=1031.655,415.008,353.471,174.280,47.465,159.655
C02629=1031.644,414.763,353.518,174.268,47.461,159.652
C02630=1031.633,414.518,353.565,174.256,47.456,159.650
C02631=1031.623,414.272,353.613,174.244,47.452,159.647
C02632=1031.612,414.027,353.659,174.233,47.447,159.644
C02633=1031.602,413.782,353.707,174.221,47.443,159.641
C02634=1031.590,413.536,353.754,174.209,47.438,159.638
C02635=1031.580,413.291,353.801,174.197,47.434,159.636
C02636=1031.569,413.046,353.847,174.185,47.429,159.633
C02637=1031.558,412.801,353.894,174.173,47.425,159.630
C02638=1031.547,412.555,353.942,174.162,47.421,159.627
C02639=1031.537,412.309,353.987,174.151,47.416,159.625
C02640=1031.526,412.064,354.035,174.139,47.412,159.622
C02641=1031.515,411.819,354.081,174.127,47.408,159.619
C02642=1031.506,411.573,354.128,174.115,47.403,159.616
C02643=1031.495,411.328,354.174,174.104,47.399,159.614
C02644=1031.485,411.082,354.221,174.093,47.395,159.611
C02645=1031.474,410.837,354.268,174.081,47.390,159.608
C02646=1031.463,410.592,354.313,174.070,47.386,159.606
C02647=1031.453,410.346,354.361,174.058,47.382,159.603
C02648=1031.442,410.101,354.407,174.047,47.377,159.600
C02649=1031.432,409.855,354.452,174.036,47.373,159.598
C02650=1031.421,409.610,354.498,174.024,47.369,159.595
C02651=1031.410,409.365,354.545,174.014,47.365,159.593
C02652=1031.400,409.119,354.591,174.002,47.361,159.590
C02653=1031.388,408.859,354.640,173.990,47.356,159.587
C02654=1031.377,408.598,354.689,173.979,47.352,159.585
C02655=1031.367,408.338,354.737,173.967,47.348,159.582
C02656=1031.356,408.077,354.785,173.955,47.344,159.579
C02657=1031.345,407.832,354.831,173.944,47.340,159.577
C02658=1031.334,407.586,354.877,173.933,47.335,159.574
C02659=1031.324,407.341,354.923,173.922,47.332,159.572
C02660=1031.314,407.096,354.969,173.912,47.328,159.569
C02661=1031.303,406.850,355.014,173.900,47.324,159.567
C02662=1031.293,406.604,355.060,173.890,47.320,159.564
C02663=1031.283,406.359,355.106,173.878,47.316,159.562
C02664=1031.273,406.113,355.152,173.868,47.312,159.559
C02665=1031.263,405.867,355.197,173.857,47.308,159.557
C02666=1031.253,405.622,355.242,173.846,47.304,159.554
C02667=1031.242,405.376,355.288,173.836,47.300,159.552
C02668=1031.232,405.131,355.333,173.825,47.297,159.549
C02669=1031.222,404.885,355.379,173.814,47.292,159.547
C02670=1031.212,404.640,355.424,173.804,47.288,159.544
C02671=1031.202,404.394,355.469,173.793,47.285,159.542
C02672=1031.192,404.148,355.515,173.782,47.281,159.540
C02673=1031.182,403.902,355.560,173.772,47.277,159.537
C02674=1031.172,403.657,355.605,173.761,47.273,159.535
C02675=1031.162,403.412,355.651,173.751,47.269,159.532
C02676=1031.152,403.166,355.696,173.740,47.266,159.530
C02677=1031.142,402.920,355.741,173.730,47.262,159.528
C02678=1031.132,402.675,355.786,173.720,47.258,159.525
C02679=1031.122,402.428,355.831,173.709,47.255,159.523
C02680=1031.112,402.183,355.876,173.699,47.251,159.521
C02681=1031.103,401.937,355.920,173.688,47.247,159.518
C02682=1031.092,401.691,355.966,173.678,47.244,159.516
C02683=1031.083,401.446,356.010,173.668,47.240,159.514
C02684=1031.073,401.200,356.055,173.658,47.236,159.512
C02685=1031.063,400.955,356.100,173.647,47.233,159.509
C02686=1031.053,400.709,356.144,173.637,47.229,159.507
C02687=1031.042,400.463,356.190,173.627,47.226,159.505
C02688=1031.033,400.217,356.234,173.617,47.222,159.502
C02689=1031.023,399.971,356.278,173.607,47.219,159.500
C02690=1031.014,399.726,356.323,173.597,47.215,159.498
C02691=1031.004,399.480,356.367,173.587,47.211,159.496
C02692=1030.994,399.235,356.412,173.577,47.208,159.494
C02693=1030.984,398.988,356.456,173.567,47.204,159.491
C02694=1030.975,398.743,356.501,173.557,47.201,159.489
C02695=1030.965,398.497,356.545,173.547,47.197,159.487
C02696=1030.955,398.252,356.589,173.537,47.194,159.485
C02697=1030.945,398.006,356.633,173.527,47.191,159.483
C02698=1030.936,397.759,356.677,173.517,47.188,159.480
C02699=1030.925,397.514,356.721,173.507,47.184,159.478
C02700=1030.916,397.268,356.765,173.497,47.181,159.476
C02701=1030.907,397.022,356.810,173.487,47.177,159.474
C02702=1030.897,396.776,356.853,173.477,47.174,159.472
C02703=1030.887,396.530,356.897,173.468,47.170,159.470
C02704=1030.877,396.284,356.942,173.459,47.167,159.468
C02705=1030.867,396.039,356.986,173.449,47.164,159.465
C02706=1030.858,395.793,357.029,173.439,47.161,159.463
C02707=1030.848,395.547,357.073,173.429,47.158,159.461
C02708=1030.839,395.301,357.117,173.419,47.155,159.459
C02709=1030.829,395.058,357.159,173.411,47.151,159.457
C02710=1030.821,394.816,357.203,173.401,47.148,159.455
C02711=1030.811,394.573,357.246,173.391,47.145,159.453
C02712=1030.801,394.331,357.289,173.382,47.141,159.451
C02713=1030.793,394.088,357.332,173.373,47.139,159.449
C02714=1030.783,393.846,357.375,173.363,47.135,159.447
C02715=1030.774,393.603,357.418,173.354,47.132,159.445
C02716=1030.764,393.361,357.461,173.345,47.129,159.443
C02717=1030.755,393.115,357.504,173.335,47.126,159.441
C02718=1030.745,392.869,357.548,173.326,47.123,159.439
C02719=1030.736,392.624,357.590,173.317,47.120,159.437
C02720=1030.727,392.377,357.634,173.307,47.117,159.435
C02721=1030.717,392.131,357.677,173.298,47.114,159.433
C02722=1030.708,391.886,357.721,173.289,47.111,159.431
C02723=1030.698,391.639,357.764,173.279,47.108,159.429
C02724=1030.690,391.393,357.807,173.270,47.105,159.427
C02725=1030.680,391.147,357.850,173.261,47.102,159.425
C02726=1030.670,390.901,357.893,173.251,47.099,159.423
C02727=1030.661,390.655,357.936,173.243,47.096,159.421
C02728=1030.652,390.410,357.979,173.233,47.093,159.419
C02729=1030.643,390.163,358.023,173.224,47.090,159.417
C02730=1030.633,389.917,358.065,173.215,47.087,159.415
C02731=1030.625,389.671,358.108,173.206,47.084,159.414
C02732=1030.615,389.425,358.151,173.197,47.081,159.412
C02733=1030.606,389.179,358.193,173.188,47.078,159.410
C02734=1030.596,388.932,358.236,173.179,47.076,159.408
C02735=1030.587,388.686,358.279,173.170,47.073,159.406
C02736=1030.578,388.441,358.321,173.161,47.070,159.404
C02737=1030.568,388.194,358.364,173.152,47.067,159.402
C02738=1030.560,387.948,358.407,173.143,47.064,159.400
C02739=1030.551,387.702,358.450,173.134,47.061,159.398
C02740=1030.541,387.456,358.493,173.125,47.059,159.397
C02741=1030.533,387.209,358.535,173.117,47.056,159.395
C02742=1030.523,386.963,358.577,173.107,47.053,159.393
C02743=1030.514,386.718,358.620,173.098,47.050,159.391
C02744=1030.504,386.471,358.662,173.089,47.048,159.389
C02745=1030.490,386.079,358.729,173.076,47.044,159.386
C02746=1030.476,385.688,358.797,173.062,47.039,159.384
C02747=1030.461,385.295,358.864,173.048,47.035,159.381
C02748=1030.446,384.904,358.930,173.034,47.031,159.378
C02749=1030.437,384.657,358.973,173.025,47.028,159.376
C02750=1030.429,384.411,359.014,173.016,47.025,159.374
C02751=1030.419,384.165,359.057,173.008,47.023,159.373
C02752=1030.410,383.919,359.099,173.000,47.020,159.371
C02753=1030.401,383.672,359.140,172.991,47.018,159.369
C02754=1030.392,383.426,359.183,172.982,47.015,159.367
C02755=1030.383,383.180,359.224,172.974,47.013,159.366
C02756=1030.374,382.934,359.266,172.965,47.010,159.364
C02757=1030.365,382.687,359.308,172.957,47.008,159.362
C02758=1030.356,382.441,359.350,172.949,47.006,159.361
C02759=1030.347,382.195,359.391,172.940,47.002,159.359
C02760=1030.339,381.948,359.433,172.932,47.000,159.357
C02761=1030.330,381.702,359.475,172.923,46.998,159.355
C02762=1030.321,381.456,359.516,172.914,46.995,159.354
C02763=1030.312,381.209,359.558,172.906,46.993,159.352
C02764=1030.303,380.963,359.600,172.898,46.990,159.350
C02765=1030.294,380.717,359.641,172.890,46.988,159.349
C02766=1030.286,380.471,359.683,172.881,46.986,159.347
C02767=1030.277,380.224,359.725,172.873,46.983,159.345
C02768=1030.268,379.978,359.766,172.865,46.981,159.344
C02769=1030.257,379.675,359.817,172.855,46.978,159.342
C02770=1030.246,379.370,359.868,172.844,46.975,159.340
C02771=1030.235,379.067,359.920,172.834,46.972,159.338
C02772=1030.225,378.764,359.970,172.824,46.969,159.336
C02773=1030.216,378.517,360.011,172.816,46.967,159.334
C02774=1030.208,378.271,360.053,172.808,46.965,159.332
C02775=1030.199,378.025,360.094,172.800,46.962,159.331
C02776=1030.190,377.778,360.135,172.792,46.960,159.329
C02777=1030.182,377.532,360.177,172.784,46.958,159.328
C02778=1030.173,377.285,360.218,172.775,46.955,159.326
C02779=1030.165,377.038,360.259,172.768,46.953,159.324
C02780=1030.156,376.793,360.299,172.759,46.951,159.323
C02781=1030.147,376.546,360.340,172.752,46.949,159.321
C02782=1030.138,376.299,360.381,172.743,46.947,159.320
C02783=1030.129,376.053,360.422,172.735,46.945,159.318
C02784=1030.121,375.806,360.463,172.728,46.943,159.317
C02785=1030.112,375.559,360.504,172.719,46.940,159.315
C02786=1030.103,375.313,360.544,172.712,46.938,159.314
C02787=1030.095,375.066,360.585,172.704,46.936,159.312
C02788=1030.087,374.820,360.626,172.696,46.934,159.311
C02789=1030.077,374.573,360.666,172.688,46.932,159.309
C02790=1030.069,374.327,360.707,172.680,46.930,159.308
C02791=1030.061,374.080,360.748,172.672,46.928,159.306
C02792=1030.052,373.834,360.788,172.664,46.926,159.305
C02793=1030.043,373.587,360.829,172.656,46.924,159.303
C02794=1030.035,373.341,360.870,172.648,46.922,159.302
C02795=1030.026,373.095,360.910,172.641,46.920,159.300
C02796=1030.018,372.848,360.951,172.633,46.918,159.299
C02797=1030.010,372.602,360.991,172.625,46.915,159.297
C02798=1030.000,372.355,361.032,172.617,46.914,159.296
C02799=1029.992,372.109,361.072,172.610,46.912,159.294
C02800=1029.985,371.862,361.112,172.602,46.910,159.293
C02801=1029.975,371.615,361.153,172.594,46.908,159.291
C02802=1029.967,371.369,361.193,172.587,46.906,159.290
C02803=1029.958,371.123,361.233,172.579,46.904,159.288
C02804=1029.950,370.875,361.274,172.572,46.902,159.287
C02805=1029.942,370.629,361.314,172.564,46.900,159.286
C02806=1029.933,370.383,361.354,172.556,46.898,159.284
C02807=1029.926,370.136,361.394,172.549,46.896,159.283
C02808=1029.917,369.889,361.435,172.541,46.895,159.281
C02809=1029.908,369.642,361.475,172.533,46.893,159.280
C02810=1029.900,369.396,361.515,172.526,46.891,159.278
C02811=1029.893,369.149,361.555,172.519,46.889,159.277
C02812=1029.884,368.903,361.595,172.511,46.887,159.276
C02813=1029.875,368.656,361.635,172.503,46.885,159.274
C02814=1029.867,368.409,361.675,172.496,46.884,159.273
C02815=1029.859,368.162,361.714,172.489,46.882,159.272
C02816=1029.850,367.917,361.754,172.481,46.880,159.270
C02817=1029.842,367.670,361.793,172.473,46.878,159.269
C02818=1029.833,367.422,361.834,172.467,46.877,159.268
C02819=1029.825,367.176,361.873,172.459,46.875,159.266
C02820=1029.816,366.929,361.912,172.451,46.873,159.265
C02821=1029.809,366.682,361.952,172.445,46.872,159.264
C02822=1029.800,366.436,361.992,172.437,46.870,159.262
C02823=1029.791,366.190,362.032,172.430,46.868,159.261
C02824=1029.784,365.943,362.072,172.423,46.866,159.259
C02825=1029.776,365.729,362.105,172.416,46.865,159.258
C02826=1029.769,365.514,362.140,172.410,46.863,159.257
C02827=1029.762,365.300,362.174,172.404,46.862,159.256
C02828=1029.755,365.086,362.208,172.397,46.861,159.255
C02829=1029.747,364.871,362.242,172.391,46.860,159.254
C02830=1029.741,364.657,362.276,172.384,46.858,159.253
C02831=1029.734,364.443,362.311,172.378,46.857,159.252
C02832=1029.726,364.229,362.345,172.371,46.855,159.250
C02833=1029.718,363.983,362.385,172.365,46.854,159.249
C02834=1029.710,363.736,362.424,172.357,46.852,159.248
C02835=1029.702,363.489,362.463,172.351,46.851,159.247
C02836=1029.694,363.242,362.502,172.343,46.849,159.245
C02837=1029.686,362.995,362.542,172.336,46.847,159.244
C02838=1029.677,362.749,362.581,172.329,46.846,159.243
C02839=1029.670,362.501,362.620,172.322,46.844,159.241
C02840=1029.662,362.255,362.659,172.315,46.843,159.240
C02841=1029.654,362.009,362.699,172.307,46.841,159.239
C02842=1029.645,361.761,362.737,172.301,46.840,159.238
C02843=1029.638,361.514,362.777,172.293,46.838,159.236
C02844=1029.629,361.267,362.816,172.286,46.837,159.235
C02845=1029.622,361.021,362.855,172.279,46.836,159.234
C02846=1029.613,360.774,362.893,172.273,46.834,159.233
C02847=1029.605,360.528,362.933,172.265,46.833,159.232
C02848=1029.598,360.280,362.972,172.259,46.831,159.230
C02849=1029.589,360.033,363.011,172.252,46.829,159.229
C02850=1029.582,359.787,363.049,172.245,46.829,159.228
C02851=1029.573,359.540,363.088,172.238,46.827,159.227
C02852=1029.565,359.292,363.127,172.231,46.826,159.226
C02853=1029.557,359.046,363.166,172.224,46.824,159.224
C02854=1029.549,358.799,363.204,172.217,46.823,159.223
C02855=1029.541,358.552,363.243,172.210,46.821,159.222
C02856=1029.533,358.305,363.281,172.203,46.821,159.221
C02857=1029.525,358.058,363.320,172.197,46.819,159.220
C02858=1029.517,357.812,363.359,172.189,46.818,159.218
C02859=1029.509,357.565,363.398,172.183,46.817,159.217
C02860=1029.501,357.318,363.435,172.176,46.815,159.216
C02861=1029.492,357.071,363.474,172.169,46.814,159.215
C02862=1029.485,356.825,363.512,172.162,46.812,159.214
C02863=1029.477,356.577,363.551,172.155,46.812,159.213
C02864=1029.469,356.330,363.589,172.149,46.810,159.212
C02865=1029.461,356.084,363.628,172.142,46.809,159.211
C02866=1029.453,355.837,363.666,172.135,46.808,159.209
C02867=1029.445,355.590,363.704,172.129,46.806,159.208
C02868=1029.437,355.342,363.742,172.122,46.805,159.207
C02869=1029.430,355.096,363.781,172.115,46.804,159.206
C02870=1029.422,354.848,363.819,172.109,46.803,159.205
C02871=1029.414,354.602,363.857,172.102,46.802,159.204
C02872=1029.405,354.355,363.895,172.095,46.801,159.203
C02873=1029.398,354.108,363.933,172.089,46.800,159.202
C02874=1029.390,353.861,363.972,172.082,46.798,159.201
C02875=1029.382,353.614,364.010,172.075,46.797,159.199
C02876=1029.374,353.367,364.047,172.069,46.796,159.198
C02877=1029.366,353.120,364.085,172.063,46.795,159.197
C02878=1029.358,352.872,364.123,172.055,46.794,159.196
C02879=1029.351,352.626,364.161,172.049,46.793,159.195
C02880=1029.343,352.379,364.198,172.042,46.792,159.194
C02881=1029.335,352.132,364.237,172.035,46.791,159.193
C02882=1029.327,351.885,364.275,172.029,46.790,159.192
C02883=1029.319,351.637,364.313,172.023,46.789,159.191
C02884=1029.311,351.391,364.350,172.017,46.788,159.190
C02885=1029.305,351.180,364.383,172.011,46.787,159.189
C02886=1029.298,350.969,364.415,172.005,46.786,159.188
C02887=1029.291,350.758,364.448,171.999,46.785,159.187
C02888=1029.285,350.546,364.479,171.994,46.784,159.186
C02889=1029.278,350.336,364.512,171.988,46.783,159.185
C02890=1029.272,350.125,364.544,171.983,46.783,159.185
C02891=1029.266,349.914,364.576,171.977,46.782,159.184
C02892=1029.259,349.703,364.608,171.972,46.781,159.183
C02893=1029.251,349.456,364.646,171.966,46.780,159.182
C02894=1029.243,349.209,364.684,171.960,46.779,159.181
C02895=1029.236,348.962,364.721,171.953,46.778,159.180
C02896=1029.228,348.715,364.758,171.946,46.777,159.179
C02897=1029.220,348.467,364.796,171.940,46.776,159.178
C02898=1029.213,348.220,364.834,171.934,46.775,159.177
C02899=1029.205,347.973,364.871,171.928,46.775,159.176
C02900=1029.198,347.726,364.908,171.921,46.774,159.175
C02901=1029.190,347.479,364.945,171.915,46.773,159.174
C02902=1029.182,347.231,364.983,171.909,46.772,159.173
C02903=1029.174,346.985,365.020,171.902,46.771,159.172
C02904=1029.167,346.738,365.058,171.896,46.770,159.171
C02905=1029.159,346.491,365.095,171.890,46.770,159.170
C02906=1029.151,346.244,365.132,171.883,46.769,159.169
C02907=1029.143,345.997,365.169,171.877,46.768,159.168
C02908=1029.136,345.750,365.207,171.871,46.767,159.167
C02909=1029.128,345.503,365.243,171.865,46.766,159.166
C02910=1029.119,345.255,365.281,171.859,46.766,159.165
C02911=1029.113,345.007,365.318,171.852,46.764,159.164
C02912=1029.105,344.761,365.354,171.846,46.764,159.163
C02913=1029.097,344.514,365.392,171.840,46.763,159.162
C02914=1029.089,344.267,365.429,171.834,46.762,159.161
C02915=1029.082,344.019,365.466,171.827,46.762,159.160
C02916=1029.074,343.772,365.503,171.821,46.761,159.159
C02917=1029.067,343.525,365.540,171.815,46.761,159.159
C02918=1029.060,343.278,365.576,171.809,46.759,159.157
C02919=1029.052,343.031,365.613,171.803,46.759,159.157
C02920=1029.044,342.784,365.651,171.797,46.759,159.156
C02921=1029.037,342.536,365.687,171.791,46.757,159.155
C02922=1029.029,342.289,365.725,171.785,46.757,159.154
C02923=1029.022,342.042,365.761,171.779,46.756,159.153
C02924=1029.014,341.795,365.797,171.773,46.756,159.152
C02925=1029.007,341.548,365.834,171.767,46.755,159.151
C02926=1028.999,341.301,365.871,171.761,46.754,159.150
C02927=1028.992,341.053,365.907,171.755,46.754,159.150
C02928=1028.984,340.806,365.945,171.749,46.753,159.149
C02929=1028.977,340.559,365.981,171.743,46.752,159.148
C02930=1028.969,340.311,366.017,171.737,46.752,159.147
C02931=1028.962,340.064,366.055,171.731,46.751,159.146
C02932=1028.955,339.818,366.091,171.725,46.751,159.145
C02933=1028.947,339.570,366.127,171.719,46.750,159.144
C02934=1028.939,339.323,366.163,171.713,46.750,159.143
C02935=1028.931,339.076,366.200,171.707,46.749,159.143
C02936=1028.924,338.828,366.236,171.701,46.749,159.142
C02937=1028.916,338.581,366.273,171.695,46.748,159.141
C02938=1028.910,338.334,366.309,171.689,46.748,159.140
C02939=1028.902,338.086,366.345,171.683,46.747,159.139
C02940=1028.894,337.839,366.381,171.677,46.747,159.138
C02941=1028.887,337.592,366.418,171.671,46.746,159.137
C02942=1028.879,337.345,366.455,171.665,46.746,159.137
C02943=1028.872,337.098,366.490,171.660,46.745,159.136
C02944=1028.864,336.851,366.527,171.654,46.745,159.135
C02945=1028.858,336.638,366.557,171.649,46.745,159.134
C02946=1028.852,336.425,366.588,171.643,46.745,159.134
C02947=1028.846,336.213,366.620,171.638,46.744,159.133
C02948=1028.839,336.000,366.651,171.634,46.744,159.132
C02949=1028.833,335.788,366.682,171.629,46.743,159.131
C02950=1028.827,335.574,366.713,171.623,46.743,159.131
C02951=1028.821,335.362,366.744,171.619,46.743,159.130
C02952=1028.813,335.150,366.775,171.614,46.742,159.129
C02953=1028.806,334.902,366.812,171.608,46.742,159.129
C02954=1028.799,334.655,366.847,171.602,46.742,159.128
C02955=1028.792,334.407,366.883,171.596,46.741,159.127
C02956=1028.785,334.160,366.919,171.590,46.741,159.126
C02957=1028.777,333.913,366.955,171.585,46.740,159.125
C02958=1028.769,333.666,366.991,171.580,46.740,159.125
C02959=1028.763,333.418,367.026,171.574,46.740,159.124
C02960=1028.755,333.171,367.063,171.568,46.740,159.123
C02961=1028.747,332.924,367.098,171.562,46.739,159.122
C02962=1028.740,332.676,367.133,171.556,46.739,159.122
C02963=1028.732,332.429,367.170,171.551,46.739,159.121
C02964=1028.725,332.182,367.205,171.545,46.738,159.120
C02965=1028.718,331.934,367.241,171.539,46.738,159.119
C02966=1028.710,331.687,367.277,171.534,46.738,159.119
C02967=1028.703,331.439,367.312,171.528,46.738,159.118
C02968=1028.695,331.193,367.348,171.523,46.737,159.117
C02969=1028.688,330.945,367.383,171.517,46.737,159.116
C02970=1028.681,330.698,367.419,171.511,46.737,159.116
C02971=1028.674,330.450,367.454,171.505,46.737,159.115
C02972=1028.667,330.203,367.489,171.501,46.737,159.114
C02973=1028.659,329.955,367.526,171.495,46.736,159.113
C02974=1028.652,329.708,367.561,171.489,46.736,159.113
C02975=1028.644,329.461,367.596,171.483,46.736,159.112
C02976=1028.637,329.213,367.632,171.478,46.736,159.111
C02977=1028.630,328.966,367.667,171.472,46.736,159.111
C02978=1028.623,328.718,367.703,171.467,46.735,159.110
C02979=1028.616,328.471,367.738,171.461,46.735,159.109
C02980=1028.609,328.224,367.773,171.456,46.735,159.108
C02981=1028.601,327.977,367.809,171.450,46.735,159.108
C02982=1028.594,327.729,367.844,171.445,46.735,159.107
C02983=1028.587,327.482,367.879,171.439,46.735,159.106
C02984=1028.579,327.234,367.914,171.434,46.735,159.106
C02985=1028.572,326.987,367.949,171.428,46.735,159.105
C02986=1028.564,326.739,367.984,171.423,46.735,159.104
C02987=1028.557,326.492,368.019,171.417,46.735,159.104
C02988=1028.550,326.245,368.054,171.412,46.734,159.103
C02989=1028.542,325.997,368.089,171.406,46.734,159.102
C02990=1028.535,325.749,368.124,171.401,46.735,159.102
C02991=1028.528,325.502,368.158,171.395,46.735,159.101
C02992=1028.520,325.254,368.194,171.389,46.735,159.100
C02993=1028.513,325.007,368.228,171.385,46.735,159.100
C02994=1028.505,324.760,368.263,171.379,46.735,159.099
C02995=1028.498,324.511,368.298,171.374,46.735,159.098
C02996=1028.491,324.264,368.332,171.368,46.735,159.098
C02997=1028.484,324.017,368.367,171.364,46.735,159.097
C02998=1028.476,323.770,368.402,171.358,46.735,159.097
C02999=1028.468,323.522,368.437,171.352,46.736,159.096
C03000=1028.461,323.275,368.472,171.347,46.736,159.095
C03001=1028.454,323.027,368.506,171.342,46.735,159.095
C03002=1028.447,322.780,368.541,171.336,46.736,159.094
C03003=1028.440,322.533,368.575,171.331,46.736,159.093
C03004=1028.432,322.284,368.610,171.325,46.736,159.093
C03005=1028.426,322.070,368.640,171.321,46.736,159.092
C03006=1028.420,321.855,368.671,171.316,46.736,159.092
C03007=1028.414,321.640,368.700,171.312,46.736,159.091
C03008=1028.408,321.426,368.730,171.307,46.736,159.090
C03009=1028.402,321.210,368.760,171.303,46.736,159.090
C03010=1028.395,320.995,368.790,171.298,46.737,159.089
C03011=1028.389,320.781,368.820,171.294,46.736,159.089
C03012=1028.383,320.566,368.850,171.289,46.737,159.088
C03013=1028.375,320.319,368.885,171.284,46.737,159.088
C03014=1028.369,320.071,368.919,171.278,46.737,159.087
C03015=1028.361,319.824,368.954,171.273,46.737,159.086
C03016=1028.354,319.576,368.987,171.268,46.738,159.086
C03017=1028.347,319.329,369.023,171.262,46.738,159.085
C03018=1028.340,319.081,369.056,171.258,46.737,159.085
C03019=1028.332,318.834,369.091,171.252,46.738,159.084
C03020=1028.326,318.586,369.125,171.247,46.738,159.084
C03021=1028.318,318.339,369.160,171.242,46.738,159.083
C03022=1028.312,318.091,369.194,171.237,46.739,159.082
C03023=1028.305,317.843,369.228,171.231,46.739,159.082
C03024=1028.297,317.596,369.263,171.227,46.739,159.081
C03025=1028.291,317.348,369.297,171.221,46.739,159.081
C03026=1028.283,317.101,369.332,171.216,46.740,159.080
C03027=1028.276,316.854,369.365,171.211,46.740,159.080
C03028=1028.270,316.606,369.400,171.206,46.740,159.079
C03029=1028.262,316.359,369.434,171.201,46.740,159.078
C03030=1028.255,316.111,369.468,171.196,46.741,159.078
C03031=1028.248,315.863,369.503,171.190,46.741,159.077
C03032=1028.242,315.616,369.536,171.186,46.741,159.077
C03033=1028.234,315.369,369.571,171.180,46.741,159.076
C03034=1028.228,315.121,369.605,171.176,46.742,159.076
C03035=1028.221,314.873,369.639,171.170,46.742,159.075
C03036=1028.214,314.625,369.673,171.165,46.742,159.074
C03037=1028.207,314.378,369.707,171.160,46.742,159.074
C03038=1028.200,314.131,369.742,171.155,46.743,159.073
C03039=1028.194,313.883,369.776,171.150,46.743,159.073
C03040=1028.186,313.636,369.810,171.145,46.744,159.072
C03041=1028.179,313.388,369.843,171.140,46.744,159.072
C03042=1028.173,313.140,369.878,171.135,46.744,159.071
C03043=1028.166,312.893,369.911,171.130,46.744,159.071
C03044=1028.159,312.645,369.945,171.125,46.745,159.070
C03045=1028.153,312.397,369.980,171.120,46.745,159.070
C03046=1028.145,312.150,370.013,171.115,46.746,159.069
C03047=1028.139,311.903,370.047,171.110,46.746,159.069
C03048=1028.132,311.655,370.081,171.105,46.746,159.068
C03049=1028.125,311.407,370.115,171.100,46.747,159.068
C03050=1028.119,311.160,370.149,171.095,46.747,159.067
C03051=1028.111,310.912,370.182,171.090,46.747,159.066
C03052=1028.104,310.665,370.216,171.086,46.748,159.066
C03053=1028.097,310.417,370.250,171.080,46.749,159.066
C03054=1028.090,310.170,370.283,171.076,46.749,159.065
C03055=1028.083,309.922,370.316,171.071,46.750,159.065
C03056=1028.075,309.674,370.350,171.065,46.750,159.064
C03057=1028.068,309.427,370.384,171.061,46.750,159.064
C03058=1028.061,309.179,370.416,171.055,46.751,159.063
C03059=1028.054,308.932,370.450,171.051,46.751,159.063
C03060=1028.047,308.683,370.483,171.046,46.752,159.062
C03061=1028.041,308.436,370.516,171.041,46.753,159.062
C03062=1028.033,308.189,370.549,171.036,46.753,159.061
C03063=1028.026,307.941,370.583,171.031,46.754,159.061
C03064=1028.019,307.694,370.616,171.027,46.755,159.060
C03065=1028.012,307.481,370.644,171.022,46.756,159.060
C03066=1028.007,307.269,370.673,171.018,46.756,159.060
C03067=1028.001,307.056,370.701,171.014,46.756,159.059
C03068=1027.995,306.844,370.729,171.009,46.757,159.059
C03069=1027.989,306.632,370.757,171.005,46.758,159.059
C03070=1027.983,306.419,370.786,171.002,46.758,159.058
C03071=1027.976,306.207,370.814,170.997,46.759,159.058
C03072=1027.971,305.994,370.843,170.993,46.759,159.057
C03073=1027.963,305.748,370.876,170.988,46.760,159.057
C03074=1027.956,305.499,370.909,170.983,46.760,159.056
C03075=1027.950,305.252,370.942,170.978,46.761,159.056
C03076=1027.942,305.004,370.975,170.974,46.762,159.056
C03077=1027.935,304.756,371.008,170.969,46.763,159.055
C03078=1027.929,304.508,371.041,170.964,46.763,159.055
C03079=1027.922,304.261,371.075,170.959,46.764,159.054
C03080=1027.915,304.014,371.107,170.955,46.765,159.054
C03081=1027.908,303.765,371.140,170.950,46.766,159.053
C03082=1027.901,303.518,371.174,170.945,46.766,159.053
C03083=1027.894,303.270,371.206,170.940,46.767,159.053
C03084=1027.887,303.023,371.239,170.936,46.767,159.052
C03085=1027.881,302.774,371.272,170.931,46.768,159.052
C03086=1027.873,302.527,371.304,170.926,46.769,159.051
C03087=1027.866,302.279,371.338,170.922,46.769,159.051
C03088=1027.860,302.032,371.371,170.917,46.770,159.050
C03089=1027.852,301.784,371.403,170.913,46.771,159.050
C03090=1027.846,301.536,371.436,170.907,46.772,159.050
C03091=1027.840,301.289,371.469,170.903,46.772,159.049
C03092=1027.832,301.041,371.501,170.898,46.774,159.049
C03093=1027.826,300.794,371.535,170.894,46.774,159.049
C03094=1027.819,300.545,371.568,170.888,46.775,159.048
C03095=1027.812,300.298,371.600,170.884,46.776,159.048
C03096=1027.805,300.051,371.633,170.880,46.776,159.047
C03097=1027.798,299.802,371.666,170.874,46.777,159.047
C03098=1027.791,299.555,371.698,170.870,46.778,159.047
C03099=1027.785,299.307,371.731,170.865,46.779,159.046
C03100=1027.778,299.059,371.764,170.861,46.780,159.046
C03101=1027.771,298.812,371.796,170.857,46.780,159.045
C03102=1027.765,298.564,371.829,170.851,46.781,159.045
C03103=1027.758,298.316,371.862,170.847,46.782,159.045
C03104=1027.751,298.069,371.894,170.842,46.783,159.044
C03105=1027.745,297.821,371.927,170.838,46.784,159.044
C03106=1027.738,297.573,371.960,170.834,46.784,159.043
C03107=1027.731,297.325,371.991,170.829,46.786,159.043
C03108=1027.725,297.077,372.024,170.824,46.786,159.043
C03109=1027.718,296.830,372.057,170.820,46.787,159.042
C03110=1027.711,296.582,372.089,170.815,46.788,159.042
C03111=1027.705,296.334,372.122,170.811,46.789,159.042
C03112=1027.698,296.087,372.155,170.806,46.789,159.041
C03113=1027.691,295.839,372.187,170.801,46.791,159.041
C03114=1027.685,295.590,372.219,170.797,46.791,159.041
C03115=1027.678,295.343,372.252,170.792,46.792,159.040
C03116=1027.671,295.095,372.284,170.788,46.793,159.040
C03117=1027.665,294.848,372.317,170.784,46.794,159.040
C03118=1027.659,294.600,372.349,170.778,46.795,159.039
C03119=1027.651,294.352,372.381,170.774,46.796,159.039
C03120=1027.645,294.104,372.414,170.770,46.797,159.039
C03121=1027.638,293.856,372.445,170.765,46.797,159.038
C03122=1027.631,293.609,372.478,170.761,46.798,159.038
C03123=1027.625,293.361,372.510,170.757,46.800,159.038
C03124=1027.618,293.113,372.542,170.752,46.800,159.037
C03125=1027.607,292.705,372.595,170.744,46.802,159.037
C03126=1027.596,292.298,372.648,170.737,46.804,159.036
C03127=1027.584,291.890,372.700,170.730,46.805,159.036
C03128=1027.573,291.482,372.752,170.723,46.807,159.035
C03129=1027.566,291.235,372.785,170.718,46.808,159.035
C03130=1027.560,290.987,372.816,170.714,46.809,159.034
C03131=1027.554,290.739,372.848,170.710,46.811,159.034
C03132=1027.547,290.492,372.880,170.705,46.812,159.034
C03133=1027.540,290.244,372.912,170.701,46.813,159.034
C03134=1027.533,289.996,372.943,170.696,46.813,159.033
C03135=1027.526,289.749,372.975,170.691,46.815,159.033
C03136=1027.519,289.500,373.007,170.687,46.816,159.033
C03137=1027.513,289.252,373.039,170.683,46.817,159.032
C03138=1027.506,289.004,373.071,170.678,46.818,159.032
C03139=1027.499,288.757,373.103,170.674,46.819,159.032
C03140=1027.492,288.509,373.134,170.670,46.820,159.032
C03141=1027.486,288.261,373.165,170.665,46.822,159.031
C03142=1027.479,288.013,373.197,170.661,46.823,159.031
C03143=1027.472,287.766,373.229,170.657,46.824,159.031
C03144=1027.466,287.517,373.261,170.652,46.825,159.030
C03145=1027.459,287.269,373.292,170.648,46.826,159.030
C03146=1027.452,287.022,373.324,170.644,46.827,159.030
C03147=1027.446,286.774,373.355,170.639,46.829,159.030
C03148=1027.439,286.526,373.387,170.635,46.830,159.029
C03149=1027.432,286.278,373.418,170.631,46.831,159.029
C03150=1027.426,286.030,373.450,170.627,46.832,159.029
C03151=1027.419,285.782,373.481,170.622,46.834,159.029
C03152=1027.412,285.534,373.512,170.618,46.835,159.028
C03153=1027.405,285.286,373.544,170.614,46.836,159.028
C03154=1027.399,285.038,373.575,170.609,46.837,159.028
C03155=1027.392,284.790,373.607,170.605,46.838,159.028
C03156=1027.385,284.543,373.638,170.601,46.839,159.027
C03157=1027.378,284.295,373.670,170.596,46.841,159.027
C03158=1027.371,284.047,373.700,170.592,46.842,159.027
C03159=1027.365,283.799,373.731,170.588,46.843,159.027
C03160=1027.358,283.551,373.763,170.584,46.845,159.026
C03161=1027.351,283.303,373.794,170.579,46.847,159.026
C03162=1027.344,283.055,373.825,170.575,46.848,159.026
C03163=1027.338,282.807,373.857,170.571,46.849,159.026
C03164=1027.331,282.559,373.888,170.566,46.850,159.025
C03165=1027.325,282.310,373.919,170.562,46.852,159.025
C03166=1027.317,282.063,373.950,170.558,46.853,159.025
C03167=1027.310,281.815,373.981,170.554,46.854,159.025
C03168=1027.304,281.568,374.012,170.550,46.856,159.025
C03169=1027.298,281.319,374.043,170.545,46.857,159.024
C03170=1027.291,281.071,374.075,170.541,46.858,159.024
C03171=1027.284,280.823,374.106,170.537,46.860,159.024
C03172=1027.278,280.575,374.137,170.533,46.861,159.024
C03173=1027.271,280.327,374.168,170.529,46.862,159.023
C03174=1027.264,280.079,374.199,170.525,46.864,159.023
C03175=1027.258,279.832,374.229,170.521,46.865,159.023
C03176=1027.251,279.584,374.261,170.516,46.866,159.023
C03177=1027.244,279.336,374.292,170.512,46.868,159.023
C03178=1027.238,279.087,374.323,170.508,46.869,159.022
C03179=1027.231,278.839,374.354,170.504,46.871,159.022
C03180=1027.225,278.592,374.385,170.499,46.872,159.022
C03181=1027.214,278.197,374.434,170.493,46.874,159.022
C03182=1027.204,277.801,374.483,170.486,46.876,159.021
C03183=1027.193,277.406,374.533,170.480,46.879,159.021
C03184=1027.183,277.011,374.582,170.473,46.881,159.021
C03185=1027.176,276.762,374.612,170.469,46.882,159.021
C03186=1027.169,276.514,374.643,170.465,46.884,159.020
C03187=1027.163,276.266,374.674,170.461,46.886,159.020
C03188=1027.156,276.018,374.704,170.456,46.887,159.020
C03189=1027.149,275.771,374.735,170.453,46.889,159.020
C03190=1027.142,275.522,374.765,170.448,46.890,159.020
C03191=1027.136,275.274,374.796,170.445,46.891,159.020
C03192=1027.130,275.027,374.827,170.441,46.893,159.020
C03193=1027.123,274.778,374.857,170.436,46.895,159.019
C03194=1027.116,274.530,374.888,170.432,46.896,159.019
C03195=1027.109,274.282,374.919,170.428,46.897,159.019
C03196=1027.103,274.034,374.949,170.424,46.899,159.019
C03197=1027.096,273.786,374.980,170.420,46.901,159.019
C03198=1027.089,273.538,375.010,170.416,46.902,159.018
C03199=1027.083,273.291,375.041,170.412,46.904,159.018
C03200=1027.076,273.042,375.071,170.408,46.905,159.018
C03201=1027.070,272.794,375.102,170.404,46.907,159.018
C03202=1027.063,272.546,375.132,170.399,46.909,159.018
C03203=1027.057,272.298,375.162,170.396,46.910,159.018
C03204=1027.049,272.050,375.192,170.392,46.912,159.018
C03205=1027.044,271.802,375.223,170.388,46.913,159.017
C03206=1027.037,271.554,375.254,170.384,46.915,159.017
C03207=1027.030,271.306,375.284,170.379,46.917,159.017
C03208=1027.024,271.058,375.315,170.376,46.918,159.017
C03209=1027.017,270.810,375.345,170.372,46.919,159.017
C03210=1027.011,270.562,375.375,170.368,46.921,159.017
C03211=1027.004,270.314,375.405,170.364,46.923,159.017
C03212=1026.997,270.065,375.436,170.360,46.925,159.017
C03213=1026.991,269.817,375.466,170.356,46.927,159.016
C03214=1026.984,269.569,375.496,170.352,46.928,159.016
C03215=1026.978,269.321,375.526,170.348,46.929,159.016
C03216=1026.971,269.073,375.556,170.344,46.931,159.016
C03217=1026.964,268.825,375.587,170.340,46.933,159.016
C03218=1026.958,268.577,375.616,170.336,46.935,159.016
C03219=1026.951,268.328,375.646,170.332,46.937,159.016
C03220=1026.944,268.081,375.676,170.328,46.938,159.016
C03221=1026.938,267.832,375.707,170.324,46.940,159.015
C03222=1026.931,267.585,375.737,170.321,46.942,159.015
C03223=1026.924,267.337,375.767,170.317,46.943,159.015
C03224=1026.918,267.088,375.797,170.312,46.945,159.015
C03225=1026.912,266.840,375.826,170.308,46.947,159.015
C03226=1026.904,266.592,375.857,170.305,46.949,159.015
C03227=1026.899,266.344,375.887,170.301,46.950,159.015
C03228=1026.891,266.096,375.917,170.297,46.952,159.015
C03229=1026.885,265.848,375.946,170.293,46.954,159.015
C03230=1026.878,265.599,375.976,170.289,46.956,159.015
C03231=1026.872,265.352,376.006,170.285,46.958,159.014
C03232=1026.865,265.103,376.037,170.281,46.959,159.014
C03233=1026.859,264.855,376.066,170.277,46.961,159.014
C03234=1026.852,264.607,376.096,170.274,46.963,159.014
C03235=1026.845,264.359,376.125,170.269,46.965,159.014
C03236=1026.838,264.111,376.155,170.265,46.966,159.014
C03237=1026.828,263.720,376.202,170.260,46.969,159.014
C03238=1026.819,263.330,376.249,170.253,46.972,159.014
C03239=1026.807,262.939,376.296,170.248,46.975,159.014
C03240=1026.798,262.548,376.342,170.241,46.978,159.013
C03241=1026.791,262.300,376.372,170.237,46.980,159.013
C03242=1026.784,262.052,376.401,170.234,46.981,159.013
C03243=1026.778,261.804,376.431,170.230,46.983,159.013
C03244=1026.771,261.555,376.461,170.226,46.985,159.013
C03245=1026.765,261.308,376.491,170.223,46.987,159.013
C03246=1026.758,261.059,376.520,170.218,46.989,159.013
C03247=1026.752,260.811,376.550,170.214,46.991,159.013
C03248=1026.746,260.563,376.579,170.210,46.993,159.013
C03249=1026.738,260.315,376.608,170.207,46.995,159.013
C03250=1026.731,260.067,376.638,170.203,46.997,159.013
C03251=1026.725,259.818,376.667,170.200,46.999,159.013
C03252=1026.718,259.570,376.696,170.195,47.001,159.013
C03253=1026.711,259.322,376.726,170.191,47.003,159.013
C03254=1026.704,259.074,376.755,170.188,47.005,159.013
C03255=1026.698,258.826,376.784,170.184,47.007,159.013
C03256=1026.691,258.577,376.813,170.180,47.009,159.013
C03257=1026.685,258.329,376.842,170.176,47.011,159.013
C03258=1026.678,258.082,376.871,170.172,47.013,159.012
C03259=1026.671,257.833,376.901,170.169,47.015,159.013
C03260=1026.664,257.585,376.930,170.165,47.017,159.012
C03261=1026.658,257.336,376.959,170.162,47.019,159.013
C03262=1026.651,257.088,376.988,170.158,47.021,159.012
C03263=1026.644,256.840,377.017,170.153,47.023,159.012
C03264=1026.638,256.591,377.046,170.150,47.025,159.012
C03265=1026.631,256.344,377.076,170.146,47.027,159.012
C03266=1026.625,256.096,377.105,170.143,47.030,159.012
C03267=1026.617,255.847,377.134,170.139,47.031,159.012
C03268=1026.611,255.599,377.163,170.135,47.034,159.012
C03269=1026.605,255.351,377.192,170.132,47.035,159.012
C03270=1026.598,255.102,377.221,170.127,47.038,159.012
C03271=1026.591,254.854,377.250,170.123,47.040,159.012
C03272=1026.585,254.606,377.279,170.120,47.042,159.012
C03273=1026.578,254.358,377.308,170.116,47.044,159.012
C03274=1026.571,254.109,377.337,170.113,47.046,159.012
C03275=1026.564,253.861,377.366,170.109,47.048,159.012
C03276=1026.558,253.613,377.395,170.106,47.050,159.012
C03277=1026.552,253.365,377.424,170.102,47.052,159.012
C03278=1026.545,253.116,377.453,170.097,47.055,159.012
C03279=1026.538,252.868,377.482,170.094,47.057,159.012
C03280=1026.532,252.620,377.511,170.090,47.059,159.012
C03281=1026.526,252.372,377.540,170.087,47.061,159.012
C03282=1026.519,252.123,377.569,170.083,47.063,159.012
C03283=1026.512,251.875,377.598,170.080,47.065,159.012
C03284=1026.506,251.627,377.627,170.076,47.067,159.012
C03285=1026.499,251.379,377.656,170.072,47.069,159.012
C03286=1026.493,251.130,377.684,170.069,47.072,159.012
C03287=1026.486,250.882,377.713,170.065,47.073,159.012
C03288=1026.480,250.634,377.742,170.061,47.076,159.012
C03289=1026.473,250.386,377.771,170.057,47.078,159.012
C03290=1026.467,250.137,377.800,170.054,47.080,159.012
C03291=1026.460,249.890,377.828,170.050,47.082,159.012
C03292=1026.454,249.642,377.857,170.046,47.084,159.012
C03293=1026.443,249.249,377.902,170.041,47.088,159.012
C03294=1026.434,248.857,377.948,170.035,47.092,159.012
C03295=1026.423,248.464,377.993,170.030,47.094,159.012
C03296=1026.413,248.072,378.039,170.023,47.098,159.012
C03297=1026.406,247.824,378.068,170.020,47.101,159.013
C03298=1026.400,247.576,378.096,170.016,47.102,159.012
C03299=1026.394,247.327,378.125,170.013,47.105,159.013
C03300=1026.387,247.080,378.154,170.009,47.107,159.013
C03301=1026.381,246.832,378.183,170.006,47.109,159.013
C03302=1026.375,246.583,378.211,170.002,47.111,159.013
C03303=1026.368,246.335,378.240,169.999,47.114,159.013
C03304=1026.362,246.087,378.269,169.995,47.115,159.013
C03305=1026.356,245.838,378.297,169.992,47.118,159.013
C03306=1026.350,245.590,378.326,169.988,47.120,159.013
C03307=1026.343,245.341,378.354,169.985,47.122,159.013
C03308=1026.337,245.093,378.383,169.981,47.124,159.013
C03309=1026.330,244.845,378.412,169.978,47.127,159.013
C03310=1026.324,244.596,378.440,169.974,47.129,159.013
C03311=1026.317,244.349,378.469,169.971,47.131,159.013
C03312=1026.311,244.101,378.498,169.967,47.133,159.013
C03313=1026.305,243.852,378.526,169.964,47.135,159.013
C03314=1026.298,243.604,378.554,169.960,47.138,159.013
C03315=1026.292,243.355,378.582,169.956,47.140,159.013
C03316=1026.286,243.107,378.610,169.952,47.143,159.013
C03317=1026.279,242.859,378.639,169.949,47.145,159.013
C03318=1026.273,242.610,378.667,169.945,47.148,159.013
C03319=1026.266,242.362,378.696,169.942,47.150,159.013
C03320=1026.260,242.114,378.724,169.938,47.152,159.013
C03321=1026.253,241.866,378.752,169.935,47.155,159.014
C03322=1026.247,241.617,378.781,169.931,47.156,159.013
C03323=1026.240,241.369,378.808,169.928,47.159,159.013
C03324=1026.233,241.121,378.837,169.924,47.161,159.014
C03325=1026.227,240.872,378.865,169.921,47.164,159.014
C03326=1026.221,240.624,378.893,169.918,47.166,159.014
C03327=1026.214,240.375,378.922,169.914,47.168,159.014
C03328=1026.208,240.127,378.950,169.911,47.171,159.014
C03329=1026.202,239.878,378.978,169.907,47.173,159.014
C03330=1026.195,239.630,379.007,169.904,47.175,159.014
C03331=1026.188,239.382,379.034,169.900,47.178,159.014
C03332=1026.181,239.134,379.062,169.896,47.181,159.014
C03333=1026.175,238.885,379.090,169.893,47.184,159.014
C03334=1026.169,238.636,379.118,169.889,47.186,159.014
C03335=1026.162,238.388,379.146,169.886,47.188,159.015
C03336=1026.155,238.140,379.174,169.882,47.191,159.015
C03337=1026.148,237.892,379.202,169.879,47.193,159.015
C03338=1026.142,237.643,379.230,169.876,47.195,159.015
C03339=1026.136,237.394,379.258,169.872,47.198,159.015
C03340=1026.130,237.147,379.285,169.869,47.201,159.015
C03341=1026.123,236.898,379.313,169.866,47.203,159.015
C03342=1026.116,236.650,379.341,169.862,47.206,159.015
C03343=1026.110,236.401,379.369,169.859,47.208,159.015
C03344=1026.103,236.153,379.396,169.855,47.210,159.015
C03345=1026.096,235.904,379.424,169.852,47.213,159.016
C03346=1026.090,235.656,379.452,169.848,47.216,159.016
C03347=1026.084,235.407,379.480,169.844,47.219,159.016
C03348=1026.077,235.159,379.508,169.841,47.221,159.016
C03349=1026.066,234.761,379.553,169.836,47.225,159.016
C03350=1026.056,234.363,379.597,169.830,47.229,159.016
C03351=1026.045,233.965,379.641,169.825,47.233,159.016
C03352=1026.035,233.566,379.686,169.819,47.238,159.017
C03353=1026.028,233.318,379.714,169.816,47.240,159.017
C03354=1026.022,233.070,379.741,169.812,47.243,159.017
C03355=1026.016,232.821,379.768,169.809,47.245,159.017
C03356=1026.009,232.572,379.796,169.806,47.248,159.017
C03357=1026.003,232.324,379.824,169.802,47.250,159.017
C03358=1025.996,232.076,379.851,169.799,47.253,159.017
C03359=1025.990,231.828,379.879,169.796,47.256,159.018
C03360=1025.984,231.579,379.907,169.792,47.258,159.018
C03361=1025.977,231.331,379.935,169.789,47.261,159.018
C03362=1025.971,231.082,379.962,169.785,47.263,159.018
C03363=1025.964,230.833,379.989,169.782,47.266,159.018
C03364=1025.958,230.585,380.017,169.779,47.268,159.018
C03365=1025.951,230.337,380.045,169.776,47.271,159.018
C03366=1025.945,230.089,380.072,169.772,47.274,159.018
C03367=1025.938,229.839,380.099,169.769,47.276,159.019
C03368=1025.932,229.592,380.127,169.766,47.279,159.019
C03369=1025.926,229.343,380.154,169.762,47.282,159.019
C03370=1025.919,229.095,380.182,169.759,47.285,159.019
C03371=1025.912,228.846,380.209,169.756,47.287,159.019
C03372=1025.906,228.598,380.236,169.752,47.289,159.019
C03373=1025.899,228.350,380.264,169.749,47.293,159.019
C03374=1025.893,228.101,380.291,169.745,47.295,159.019
C03375=1025.886,227.852,380.318,169.742,47.298,159.020
C03376=1025.880,227.605,380.346,169.738,47.301,159.020
C03377=1025.874,227.356,380.373,169.735,47.304,159.020
C03378=1025.867,227.107,380.401,169.732,47.306,159.020
C03379=1025.861,226.859,380.427,169.729,47.309,159.020
C03380=1025.854,226.611,380.454,169.725,47.312,159.020
C03381=1025.847,226.362,380.482,169.722,47.315,159.021
C03382=1025.841,226.113,380.509,169.719,47.318,159.021
C03383=1025.834,225.866,380.536,169.715,47.320,159.021
C03384=1025.827,225.617,380.563,169.712,47.323,159.021
C03385=1025.821,225.368,380.591,169.709,47.325,159.021
C03386=1025.815,225.120,380.617,169.706,47.328,159.022
C03387=1025.808,224.871,380.644,169.703,47.332,159.022
C03388=1025.801,224.623,380.671,169.699,47.334,159.022
C03389=1025.795,224.374,380.698,169.696,47.337,159.022
C03390=1025.788,224.126,380.725,169.693,47.339,159.022
C03391=1025.782,223.877,380.752,169.689,47.342,159.023
C03392=1025.776,223.629,380.780,169.685,47.346,159.023
C03393=1025.768,223.381,380.806,169.682,47.348,159.023
C03394=1025.762,223.132,380.833,169.679,47.351,159.023
C03395=1025.756,222.884,380.860,169.676,47.354,159.023
C03396=1025.750,222.635,380.887,169.672,47.357,159.023
C03397=1025.742,222.387,380.914,169.669,47.360,159.024
C03398=1025.736,222.138,380.941,169.666,47.363,159.024
C03399=1025.730,221.889,380.968,169.663,47.365,159.024
C03400=1025.723,221.642,380.995,169.659,47.368,159.024
C03401=1025.717,221.393,381.022,169.656,47.371,159.024
C03402=1025.710,221.144,381.049,169.653,47.374,159.024
C03403=1025.704,220.896,381.076,169.650,47.377,159.025
C03404=1025.697,220.647,381.103,169.647,47.380,159.025
C03405=1025.687,220.241,381.147,169.641,47.384,159.025
C03406=1025.676,219.835,381.191,169.636,47.389,159.026
C03407=1025.666,219.429,381.234,169.630,47.394,159.026
C03408=1025.655,219.023,381.278,169.626,47.399,159.026
C03409=1025.649,218.774,381.305,169.622,47.401,159.026
C03410=1025.642,218.526,381.332,169.619,47.404,159.027
C03411=1025.636,218.278,381.358,169.616,47.407,159.027
C03412=1025.629,218.029,381.385,169.613,47.410,159.027
C03413=1025.623,217.781,381.412,169.609,47.414,159.027
C03414=1025.616,217.532,381.438,169.606,47.417,159.028
C03415=1025.609,217.284,381.464,169.603,47.420,159.028
C03416=1025.603,217.035,381.491,169.600,47.423,159.028
C03417=1025.597,216.787,381.517,169.596,47.426,159.028
C03418=1025.590,216.538,381.544,169.593,47.428,159.028
C03419=1025.583,216.289,381.571,169.590,47.431,159.029
C03420=1025.576,216.041,381.597,169.587,47.434,159.029
C03421=1025.570,215.792,381.624,169.584,47.437,159.029
C03422=1025.563,215.544,381.650,169.581,47.441,159.029
C03423=1025.557,215.295,381.677,169.577,47.444,159.030
C03424=1025.550,215.047,381.703,169.574,47.447,159.030
C03425=1025.543,214.798,381.730,169.571,47.450,159.030
C03426=1025.538,214.550,381.757,169.568,47.453,159.030
C03427=1025.530,214.301,381.783,169.565,47.456,159.031
C03428=1025.525,214.053,381.810,169.562,47.459,159.031
C03429=1025.518,213.804,381.835,169.559,47.462,159.031
C03430=1025.511,213.556,381.861,169.556,47.465,159.031
C03431=1025.506,213.307,381.888,169.553,47.468,159.032
C03432=1025.499,213.058,381.914,169.549,47.471,159.032
C03433=1025.493,212.810,381.941,169.546,47.474,159.032
C03434=1025.486,212.561,381.967,169.542,47.478,159.032
C03435=1025.479,212.313,381.994,169.539,47.481,159.032
C03436=1025.473,212.064,382.021,169.536,47.484,159.033
C03437=1025.466,211.816,382.047,169.533,47.487,159.033
C03438=1025.459,211.567,382.073,169.530,47.490,159.033
C03439=1025.453,211.319,382.100,169.527,47.493,159.033
C03440=1025.447,211.071,382.126,169.523,47.496,159.034
C03441=1025.441,210.821,382.152,169.520,47.499,159.034
C03442=1025.434,210.573,382.178,169.517,47.502,159.034
C03443=1025.427,210.325,382.204,169.514,47.505,159.034
C03444=1025.421,210.077,382.231,169.511,47.508,159.035
C03445=1025.415,209.828,382.257,169.508,47.511,159.035
C03446=1025.408,209.579,382.283,169.505,47.514,159.035
C03447=1025.402,209.331,382.309,169.502,47.518,159.035
C03448=1025.394,209.082,382.335,169.499,47.521,159.036
C03449=1025.388,208.834,382.361,169.496,47.524,159.036
C03450=1025.382,208.585,382.387,169.493,47.527,159.036
C03451=1025.375,208.336,382.414,169.490,47.531,159.037
C03452=1025.369,208.088,382.440,169.486,47.534,159.037
C03453=1025.362,207.839,382.466,169.483,47.537,159.037
C03454=1025.355,207.591,382.492,169.480,47.540,159.037
C03455=1025.349,207.343,382.518,169.477,47.543,159.038
C03456=1025.343,207.093,382.544,169.474,47.547,159.038
C03457=1025.336,206.845,382.570,169.471,47.550,159.038
C03458=1025.330,206.597,382.596,169.468,47.553,159.039
C03459=1025.323,206.348,382.622,169.465,47.556,159.039
C03460=1025.317,206.100,382.648,169.461,47.560,159.039
C03461=1025.306,205.696,382.690,169.457,47.565,159.039
C03462=1025.295,205.292,382.732,169.451,47.571,159.040
C03463=1025.285,204.890,382.774,169.447,47.576,159.040
C03464=1025.274,204.487,382.815,169.442,47.581,159.041
C03465=1025.250,203.453,382.916,169.042,47.480,158.967
C03466=1025.244,203.204,382.941,169.038,47.484,158.967
C03467=1025.239,202.955,382.965,169.035,47.488,158.968
C03468=1025.233,202.706,382.990,169.030,47.492,158.968
C03469=1025.227,202.458,383.015,169.026,47.496,158.968
C03470=1025.221,202.209,383.039,169.022,47.500,158.969
C03471=1025.215,201.960,383.063,169.018,47.504,158.969
C03472=1025.210,201.712,383.087,169.013,47.508,158.969
C03473=1025.204,201.462,383.112,169.010,47.513,158.970
C03474=1025.198,201.214,383.136,169.006,47.517,158.970
C03475=1025.193,200.966,383.160,169.002,47.521,158.970
C03476=1025.187,200.716,383.184,168.998,47.525,158.971
C03477=1025.182,200.468,383.209,168.994,47.529,158.971
C03478=1025.176,200.218,383.233,168.990,47.533,158.971
C03479=1025.170,199.970,383.257,168.986,47.537,158.972
C03480=1025.164,199.722,383.281,168.982,47.541,158.972
C03481=1025.158,199.473,383.305,168.978,47.546,158.972
C03482=1025.153,199.223,383.329,168.973,47.550,158.973
C03483=1025.146,198.974,383.353,168.970,47.554,158.973
C03484=1025.141,198.726,383.377,168.966,47.559,158.973
C03485=1025.135,198.478,383.401,168.962,47.563,158.974
C03486=1025.128,198.229,383.425,168.957,47.568,158.974
C03487=1025.123,197.979,383.448,168.954,47.572,158.974
C03488=1025.117,197.731,383.472,168.950,47.576,158.975
C03489=1025.111,197.482,383.497,168.946,47.580,158.975
C03490=1025.105,197.234,383.520,168.942,47.584,158.975
C03491=1025.099,196.985,383.543,168.938,47.589,158.976
C03492=1025.093,196.735,383.568,168.934,47.593,158.976
C03493=1025.087,196.487,383.592,168.930,47.597,158.976
C03494=1025.082,196.238,383.616,168.926,47.601,158.977
C03495=1025.076,195.990,383.639,168.923,47.606,158.977
C03496=1025.070,195.740,383.663,168.918,47.610,158.978
C03497=1025.064,195.492,383.687,168.914,47.614,158.978
C03498=1025.059,195.243,383.710,168.911,47.619,158.978
C03499=1025.053,194.995,383.734,168.907,47.623,158.979
C03500=1025.047,194.745,383.758,168.903,47.627,158.979
C03501=1025.042,194.496,383.782,168.899,47.632,158.980
C03502=1025.036,194.248,383.805,168.895,47.636,158.980
C03503=1025.030,193.999,383.828,168.891,47.640,158.980
C03504=1025.024,193.750,383.853,168.887,47.645,158.981
C03505=1025.018,193.502,383.877,168.883,47.649,158.981
C03506=1025.013,193.252,383.900,168.880,47.653,158.981
C03507=1025.007,193.004,383.924,168.876,47.658,158.982
C03508=1025.001,192.755,383.947,168.872,47.662,158.982
C03509=1024.995,192.506,383.971,168.867,47.666,158.982
C03510=1024.990,192.257,383.994,168.864,47.671,158.983
C03511=1024.984,192.009,384.018,168.860,47.675,158.983
C03512=1024.979,191.760,384.042,168.856,47.679,158.983
C03513=1024.973,191.511,384.065,168.853,47.684,158.984
C03514=1024.967,191.261,384.089,168.849,47.688,158.984
C03515=1024.961,191.013,384.113,168.845,47.692,158.985
C03516=1024.955,190.764,384.136,168.842,47.696,158.985
C03517=1024.950,190.516,384.160,168.838,47.700,158.985
C03518=1024.944,190.267,384.183,168.834,47.705,158.986
C03519=1024.939,190.018,384.207,168.829,47.710,158.986
C03520=1024.933,189.769,384.230,168.825,47.714,158.986
C03521=1024.927,189.521,384.254,168.822,47.718,158.987
C03522=1024.922,189.271,384.278,168.818,47.722,158.987
C03523=1024.916,189.022,384.301,168.814,47.726,158.988
C03524=1024.910,188.774,384.324,168.811,47.731,158.988
C03525=1024.905,188.525,384.348,168.807,47.735,158.988
C03526=1024.898,188.243,384.374,168.802,47.740,158.989
C03527=1024.892,187.960,384.401,168.799,47.745,158.989
C03528=1024.886,187.677,384.428,168.794,47.750,158.990
C03529=1024.879,187.395,384.454,168.790,47.755,158.990
C03530=1024.874,187.146,384.477,168.786,47.759,158.990
C03531=1024.868,186.898,384.501,168.783,47.764,158.991
C03532=1024.863,186.649,384.524,168.779,47.768,158.991
C03533=1024.858,186.400,384.548,168.775,47.772,158.991
C03534=1024.852,186.151,384.571,168.771,47.777,158.992
C03535=1024.846,185.902,384.594,168.768,47.781,158.992
C03536=1024.841,185.653,384.618,168.764,47.785,158.993
C03537=1024.835,185.405,384.641,168.760,47.789,158.993
C03538=1024.829,185.156,384.664,168.756,47.793,158.993
C03539=1024.824,184.907,384.688,168.753,47.798,158.994
C03540=1024.818,184.658,384.711,168.749,47.802,158.994
C03541=1024.813,184.409,384.734,168.746,47.807,158.995
C03542=1024.807,184.160,384.758,168.742,47.811,158.995
C03543=1024.802,183.912,384.781,168.738,47.815,158.995
C03544=1024.796,183.663,384.804,168.734,47.820,158.996
C03545=1024.791,183.413,384.828,168.731,47.824,158.996
C03546=1024.785,183.165,384.851,168.727,47.829,158.997
C03547=1024.780,182.915,384.874,168.724,47.832,158.997
C03548=1024.774,182.667,384.898,168.720,47.836,158.997
C03549=1024.768,182.418,384.921,168.717,47.841,158.998
C03550=1024.763,182.169,384.943,168.712,47.846,158.998
C03551=1024.757,181.920,384.966,168.709,47.850,158.999
C03552=1024.751,181.671,384.988,168.705,47.855,158.999
C03553=1024.745,181.422,385.011,168.702,47.860,159.000
C03554=1024.739,181.173,385.034,168.698,47.865,159.000
C03555=1024.734,180.925,385.057,168.694,47.869,159.000
C03556=1024.727,180.676,385.079,168.691,47.873,159.001
C03557=1024.721,180.427,385.102,168.687,47.878,159.001
C03558=1024.716,180.178,385.125,168.684,47.883,159.002
C03559=1024.710,179.929,385.147,168.680,47.887,159.002
C03560=1024.704,179.680,385.170,168.677,47.892,159.003
C03561=1024.698,179.431,385.193,168.673,47.896,159.003
C03562=1024.692,179.182,385.216,168.670,47.901,159.004
C03563=1024.687,178.933,385.238,168.666,47.905,159.004
C03564=1024.680,178.684,385.260,168.662,47.910,159.004
C03565=1024.675,178.435,385.283,168.659,47.915,159.005
C03566=1024.669,178.186,385.306,168.655,47.919,159.005
C03567=1024.663,177.937,385.328,168.651,47.924,159.006
C03568=1024.657,177.688,385.351,168.648,47.928,159.006
C03569=1024.652,177.440,385.373,168.644,47.933,159.007
C03570=1024.646,177.191,385.396,168.641,47.938,159.007
C03571=1024.640,176.942,385.418,168.637,47.942,159.007
C03572=1024.634,176.693,385.441,168.634,47.947,159.008
C03573=1024.629,176.444,385.464,168.630,47.951,159.008
C03574=1024.623,176.195,385.486,168.627,47.956,159.009
C03575=1024.617,175.946,385.508,168.623,47.960,159.009
C03576=1024.611,175.697,385.531,168.619,47.965,159.010
C03577=1024.606,175.448,385.553,168.616,47.970,159.010
C03578=1024.600,175.200,385.576,168.612,47.974,159.011
C03579=1024.594,174.951,385.599,168.609,47.979,159.011
C03580=1024.589,174.701,385.621,168.605,47.983,159.011
C03581=1024.583,174.452,385.644,168.602,47.988,159.012
C03582=1024.577,174.203,385.665,168.598,47.993,159.012
C03583=1024.572,173.955,385.688,168.594,47.997,159.013
C03584=1024.566,173.706,385.711,168.591,48.002,159.013
C03585=1024.560,173.457,385.732,168.587,48.006,159.014
C03586=1024.554,173.208,385.755,168.584,48.011,159.014
C03587=1024.548,172.959,385.778,168.580,48.016,159.015
C03588=1024.543,172.710,385.800,168.576,48.020,159.015
C03589=1024.537,172.461,385.822,168.573,48.025,159.015
C03590=1024.531,172.178,385.848,168.570,48.030,159.016
C03591=1024.525,171.896,385.874,168.565,48.035,159.016
C03592=1024.518,171.612,385.898,168.562,48.040,159.017
C03593=1024.512,171.330,385.924,168.558,48.046,159.018
C03594=1024.506,171.080,385.946,168.554,48.051,159.018
C03595=1024.500,170.832,385.969,168.550,48.055,159.018
C03596=1024.495,170.583,385.990,168.547,48.059,159.019
C03597=1024.489,170.334,386.013,168.544,48.064,159.019
C03598=1024.483,170.085,386.035,168.541,48.069,159.020
C03599=1024.477,169.836,386.058,168.537,48.073,159.020
C03600=1024.472,169.587,386.080,168.534,48.078,159.021
C03601=1024.466,169.338,386.101,168.530,48.082,159.021
C03602=1024.461,169.089,386.124,168.527,48.087,159.022
C03603=1024.456,168.840,386.146,168.523,48.091,159.022
C03604=1024.450,168.591,386.169,168.519,48.096,159.022
C03605=1024.444,168.342,386.191,168.517,48.101,159.023
C03606=1024.439,168.093,386.213,168.513,48.105,159.023
C03607=1024.433,167.844,386.236,168.510,48.110,159.024
C03608=1024.427,167.595,386.257,168.506,48.114,159.024
C03609=1024.422,167.347,386.280,168.503,48.119,159.025
C03610=1024.417,167.097,386.302,168.499,48.124,159.025
C03611=1024.410,166.848,386.324,168.497,48.128,159.026
C03612=1024.405,166.600,386.346,168.493,48.132,159.026
C03613=1024.400,166.350,386.369,168.489,48.137,159.026
C03614=1024.394,166.101,386.390,168.486,48.142,159.027
C03615=1024.389,165.853,386.413,168.483,48.147,159.027
C03616=1024.383,165.604,386.435,168.479,48.152,159.028
C03617=1024.378,165.355,386.456,168.476,48.155,159.028
C03618=1024.372,165.106,386.478,168.473,48.160,159.029
C03619=1024.366,164.857,386.501,168.469,48.165,159.029
C03620=1024.361,164.608,386.523,168.466,48.170,159.030
C03621=1024.355,164.359,386.545,168.462,48.174,159.030
C03622=1024.350,164.110,386.567,168.460,48.178,159.031
C03623=1024.344,163.861,386.589,168.456,48.183,159.031
C03624=1024.339,163.612,386.611,168.453,48.188,159.032
C03625=1024.334,163.363,386.633,168.449,48.192,159.032
C03626=1024.328,163.114,386.655,168.446,48.197,159.032
C03627=1024.323,162.865,386.677,168.443,48.201,159.033
C03628=1024.317,162.616,386.700,168.439,48.206,159.033
C03629=1024.312,162.367,386.721,168.436,48.211,159.034
